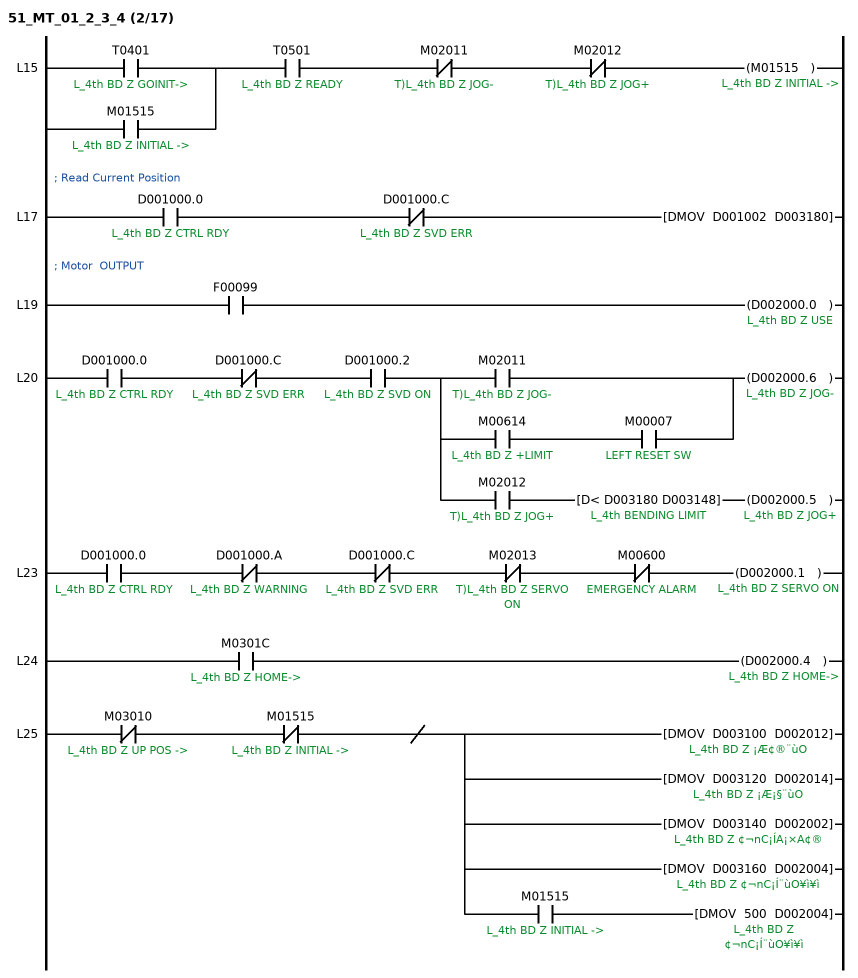
[picture p240: 51_MT_01_2_3_4 rungs L15-L25]
; L15
LOAD      T0401	// L_4th BD Z GOINIT->
OR        M01515	// L_4th BD Z INITIAL ->
AND       T0501	// L_4th BD Z READY
AND NOT   M02011	// T)L_4th BD Z JOG-
AND NOT   M02012	// T)L_4th BD Z JOG+
OUT       M01515	// L_4th BD Z INITIAL ->
; L17
LOAD      D001000.0	// L_4th BD Z CTRL RDY
AND NOT   D001000.C	// L_4th BD Z SVD ERR
DMOV      D001002 D003180
// output comment: Read Current Position
//  Motor  OUTPUT
; L19
LOAD      F00099
OUT       D002000.0	// L_4th BD Z USE
; L20
LOAD      D001000.0	// L_4th BD Z CTRL RDY
AND NOT   D001000.C	// L_4th BD Z SVD ERR
AND       D001000.2	// L_4th BD Z SVD ON
MPUSH
LOAD      M02011	// T)L_4th BD Z JOG-
LOAD      M00614	// L_4th BD Z +LIMIT
AND       M00007	// LEFT RESET SW
OR LOAD
AND LOAD
OUT       D002000.6	// L_4th BD Z JOG-
MPOP
AND       M02012	// T)L_4th BD Z JOG+
ANDD<     D003180 D003148	// L_4th BENDING LIMIT
OUT       D002000.5	// L_4th BD Z JOG+
; L23
LOAD      D001000.0	// L_4th BD Z CTRL RDY
AND NOT   D001000.A	// L_4th BD Z WARNING
AND NOT   D001000.C	// L_4th BD Z SVD ERR
AND NOT   M02013	// T)L_4th BD Z SERVO ON
AND NOT   M00600	// EMERGENCY ALARM
OUT       D002000.1	// L_4th BD Z SERVO ON
; L24
LOAD      M0301C	// L_4th BD Z HOME->
OUT       D002000.4	// L_4th BD Z HOME->
; L25
LOAD NOT  M03010	// L_4th BD Z UP POS ->
AND NOT   M01515	// L_4th BD Z INITIAL ->
NOT
DMOV      D003100 D002012	// L_4th BD Z ¡Æ¢®¨ùO
DMOV      D003120 D002014	// L_4th BD Z ¡Æ¡§¨ùO
DMOV      D003140 D002002	// L_4th BD Z ¢¬nC¡ÍA¡×A¢®
DMOV      D003160 D002004	// L_4th BD Z ¢¬nC¡Í¨ùO¥ì¥ì
AND       M01515	// L_4th BD Z INITIAL ->
DMOV      500 D002004	// L_4th BD Z ¢¬nC¡Í¨ùO¥ì¥ì

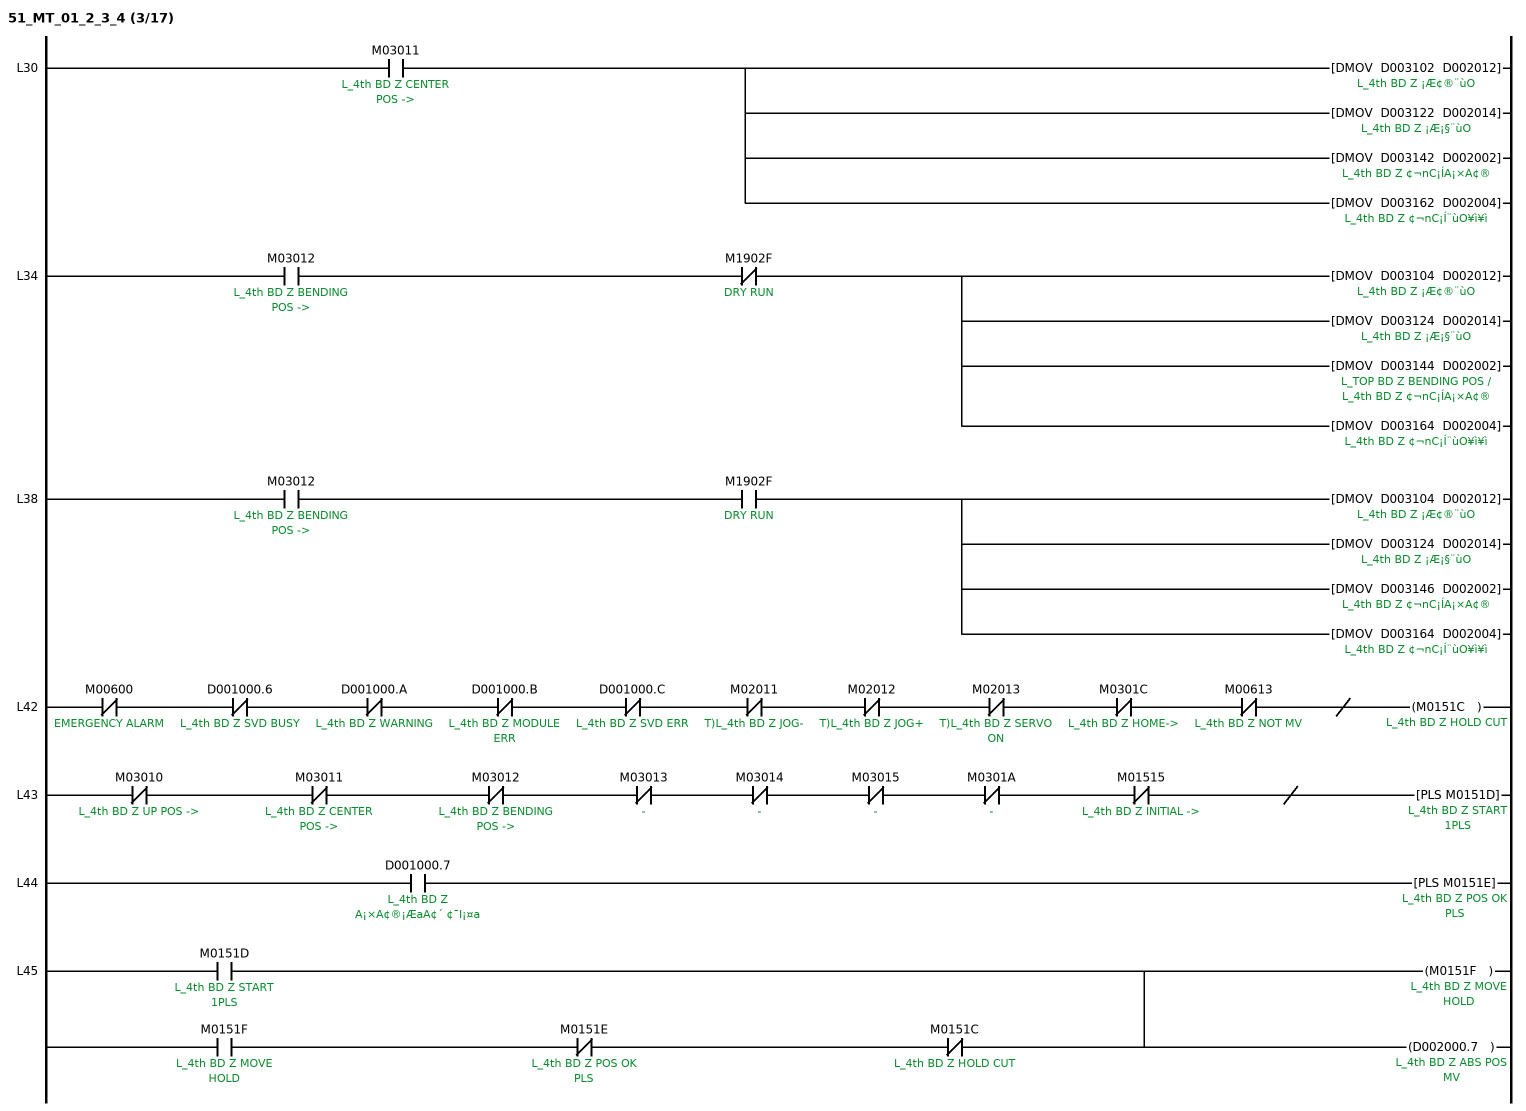
; L30
LOAD      M03011	// L_4th BD Z CENTER POS ->
DMOV      D003102 D002012	// L_4th BD Z ¡Æ¢®¨ùO
DMOV      D003122 D002014	// L_4th BD Z ¡Æ¡§¨ùO
DMOV      D003142 D002002	// L_4th BD Z ¢¬nC¡ÍA¡×A¢®
DMOV      D003162 D002004	// L_4th BD Z ¢¬nC¡Í¨ùO¥ì¥ì
; L34
LOAD      M03012	// L_4th BD Z BENDING POS ->
AND NOT   M1902F	// DRY RUN
DMOV      D003104 D002012	// L_4th BD Z ¡Æ¢®¨ùO
DMOV      D003124 D002014	// L_4th BD Z ¡Æ¡§¨ùO
DMOV      D003144 D002002	// L_TOP BD Z BENDING POS / L_4th BD Z ¢¬nC¡ÍA¡×A¢®
DMOV      D003164 D002004	// L_4th BD Z ¢¬nC¡Í¨ùO¥ì¥ì
; L38
LOAD      M03012	// L_4th BD Z BENDING POS ->
AND       M1902F	// DRY RUN
DMOV      D003104 D002012	// L_4th BD Z ¡Æ¢®¨ùO
DMOV      D003124 D002014	// L_4th BD Z ¡Æ¡§¨ùO
DMOV      D003146 D002002	// L_4th BD Z ¢¬nC¡ÍA¡×A¢®
DMOV      D003164 D002004	// L_4th BD Z ¢¬nC¡Í¨ùO¥ì¥ì
; L42
LOAD NOT  M00600	// EMERGENCY ALARM
AND NOT   D001000.6	// L_4th BD Z SVD BUSY
AND NOT   D001000.A	// L_4th BD Z WARNING
AND NOT   D001000.B	// L_4th BD Z MODULE ERR
AND NOT   D001000.C	// L_4th BD Z SVD ERR
AND NOT   M02011	// T)L_4th BD Z JOG-
AND NOT   M02012	// T)L_4th BD Z JOG+
AND NOT   M02013	// T)L_4th BD Z SERVO ON
AND NOT   M0301C	// L_4th BD Z HOME->
AND NOT   M00613	// L_4th BD Z NOT MV
NOT
OUT       M0151C	// L_4th BD Z HOLD CUT
; L43
LOAD NOT  M03010	// L_4th BD Z UP POS ->
AND NOT   M03011	// L_4th BD Z CENTER POS ->
AND NOT   M03012	// L_4th BD Z BENDING POS ->
AND NOT   M03013	// -
AND NOT   M03014	// -
AND NOT   M03015	// -
AND NOT   M0301A	// -
AND NOT   M01515	// L_4th BD Z INITIAL ->
NOT
OUTP      M0151D	// L_4th BD Z START 1PLS
; L44
LOAD      D001000.7	// L_4th BD Z A¡×A¢®¡ÆaA¢´ ¢¯I¡¤a
OUTP      M0151E	// L_4th BD Z POS OK PLS
; L45
LOAD      M0151D	// L_4th BD Z START 1PLS
LOAD      M0151F	// L_4th BD Z MOVE HOLD
AND NOT   M0151E	// L_4th BD Z POS OK PLS
AND NOT   M0151C	// L_4th BD Z HOLD CUT
OR LOAD
OUT       M0151F	// L_4th BD Z MOVE HOLD
OUT       D002000.7	// L_4th BD Z ABS POS MV

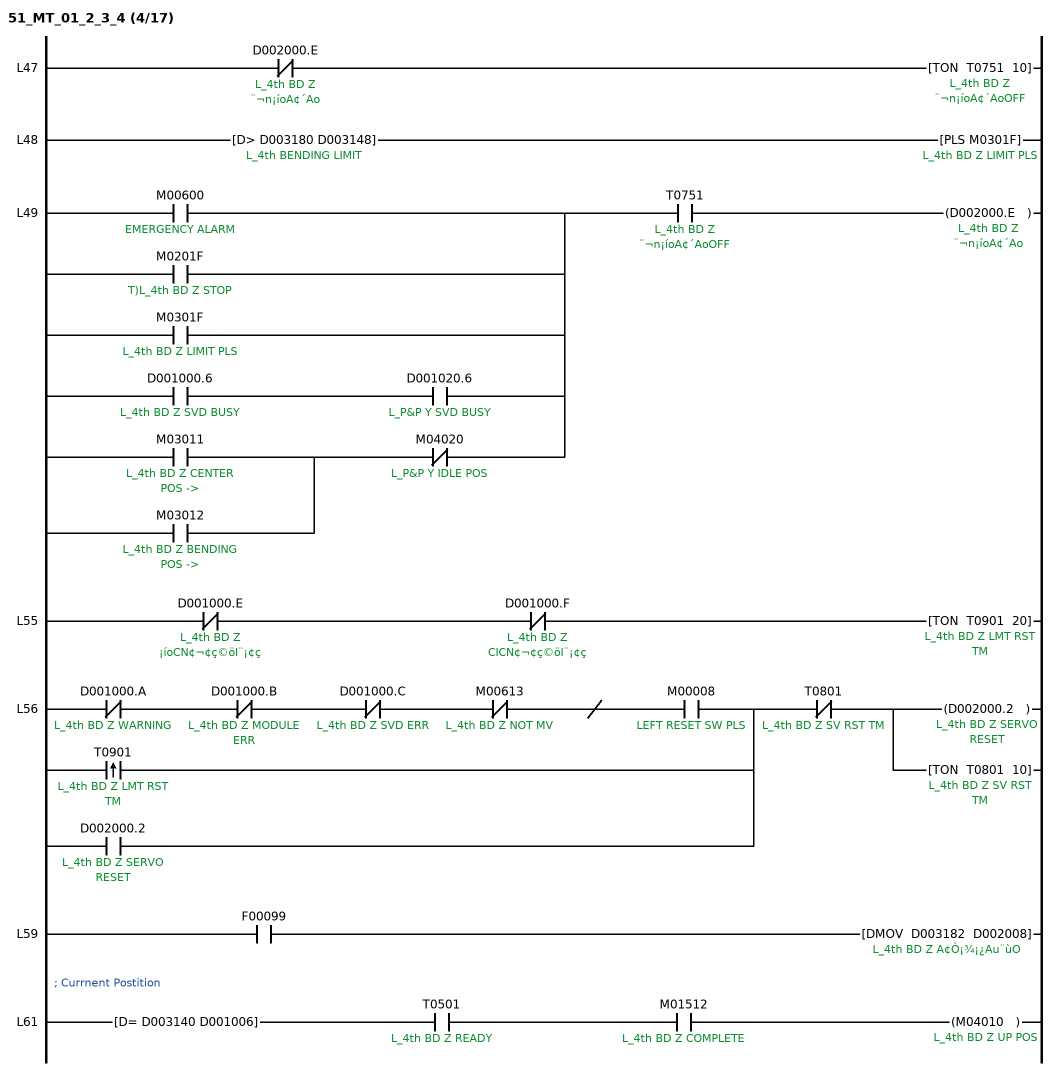
; L47
LOAD NOT  D002000.E	// L_4th BD Z ¨¬n¡íoA¢´Ao
TON       T0751 10	// L_4th BD Z ¨¬n¡íoA¢´AoOFF
; L48
LOADD>    D003180 D003148	// L_4th BENDING LIMIT
OUTP      M0301F	// L_4th BD Z LIMIT PLS
; L49
LOAD      M00600	// EMERGENCY ALARM
OR        M0201F	// T)L_4th BD Z STOP
OR        M0301F	// L_4th BD Z LIMIT PLS
LOAD      D001000.6	// L_4th BD Z SVD BUSY
AND       D001020.6	// L_P&P Y SVD BUSY
OR LOAD
LOAD      M03011	// L_4th BD Z CENTER POS ->
OR        M03012	// L_4th BD Z BENDING POS ->
AND NOT   M04020	// L_P&P Y IDLE POS
OR LOAD
AND       T0751	// L_4th BD Z ¨¬n¡íoA¢´AoOFF
OUT       D002000.E	// L_4th BD Z ¨¬n¡íoA¢´Ao
; L55
LOAD NOT  D001000.E	// L_4th BD Z ¡íoCN¢¬¢ç©öI¨¡¢ç
AND NOT   D001000.F	// L_4th BD Z CICN¢¬¢ç©öI¨¡¢ç
TON       T0901 20	// L_4th BD Z LMT RST TM
; L56
LOAD NOT  D001000.A	// L_4th BD Z WARNING
AND NOT   D001000.B	// L_4th BD Z MODULE ERR
AND NOT   D001000.C	// L_4th BD Z SVD ERR
AND NOT   M00613	// L_4th BD Z NOT MV
NOT
AND       M00008	// LEFT RESET SW PLS
ORP       T0901	// L_4th BD Z LMT RST TM
OR        D002000.2	// L_4th BD Z SERVO RESET
AND NOT   T0801	// L_4th BD Z SV RST TM
OUT       D002000.2	// L_4th BD Z SERVO RESET
TON       T0801 10	// L_4th BD Z SV RST TM
; L59
LOAD      F00099
DMOV      D003182 D002008	// L_4th BD Z A¢Ò¡¾¡¿Au¨ùO
// Currnent Postition
; L61
LOADD=    D003140 D001006
AND       T0501	// L_4th BD Z READY
AND       M01512	// L_4th BD Z COMPLETE
OUT       M04010	// L_4th BD Z UP POS

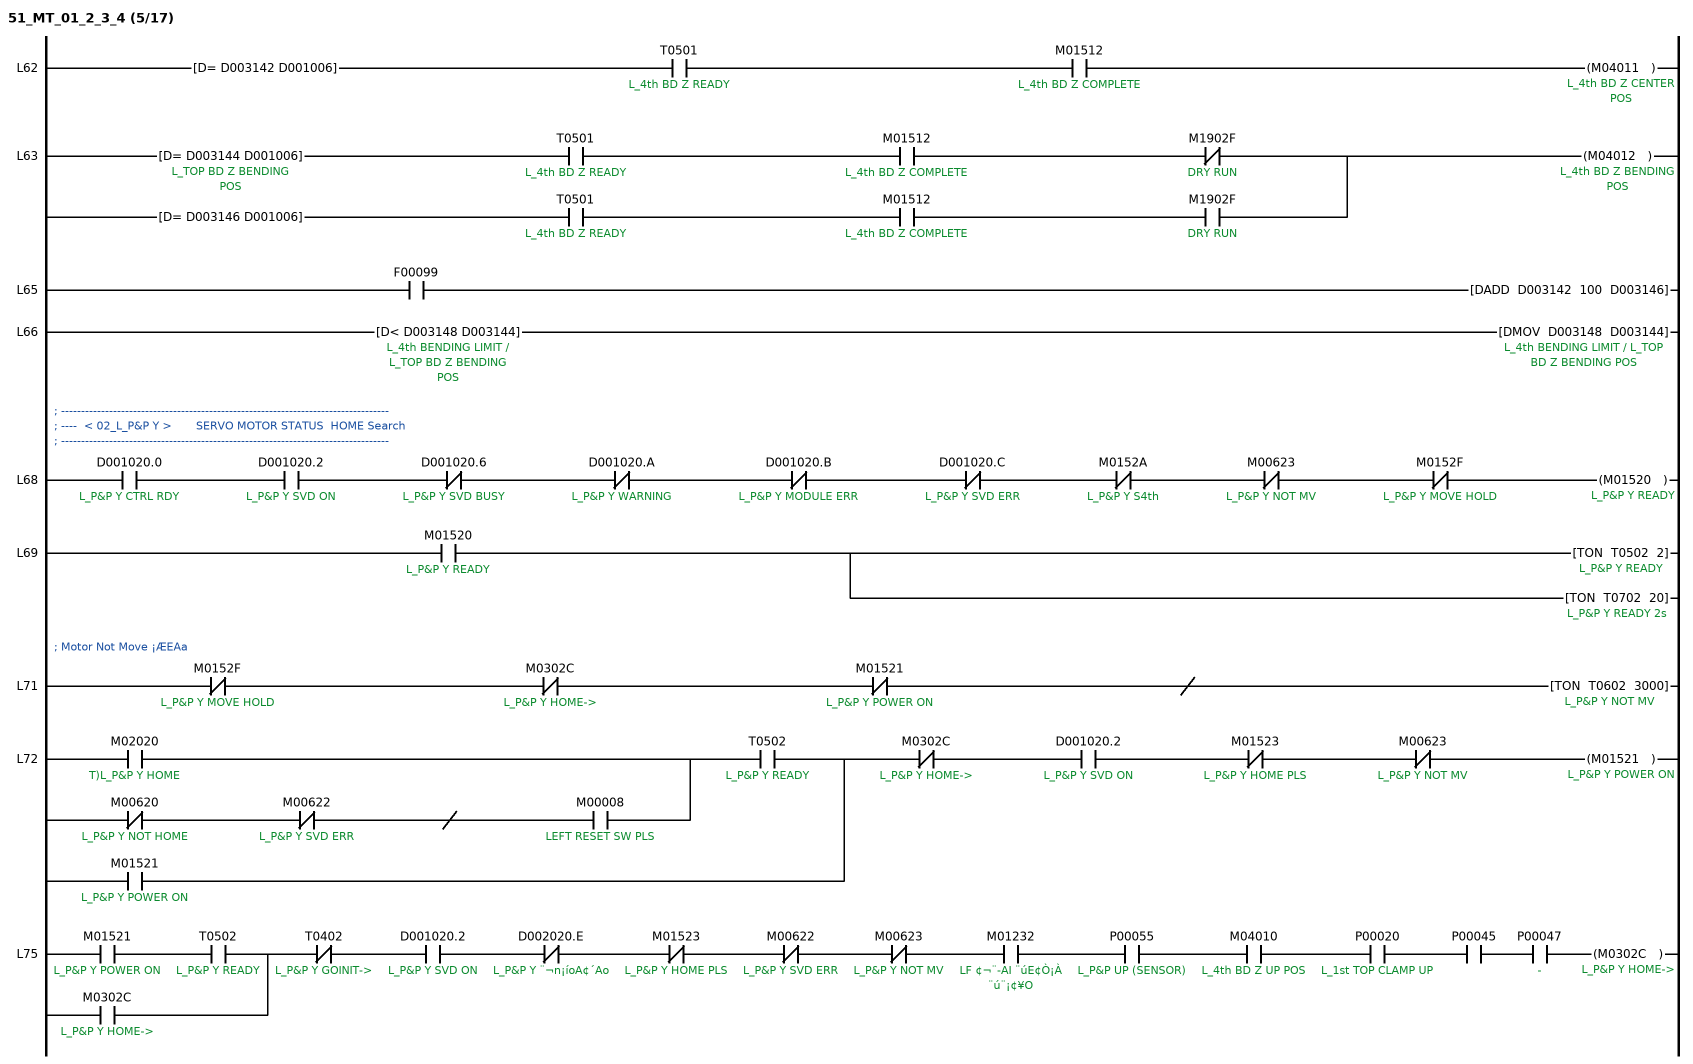
; L62
LOADD=    D003142 D001006
AND       T0501	// L_4th BD Z READY
AND       M01512	// L_4th BD Z COMPLETE
OUT       M04011	// L_4th BD Z CENTER POS
; L63
LOADD=    D003144 D001006	// L_TOP BD Z BENDING POS
AND       T0501	// L_4th BD Z READY
AND       M01512	// L_4th BD Z COMPLETE
AND NOT   M1902F	// DRY RUN
LOADD=    D003146 D001006
AND       T0501	// L_4th BD Z READY
AND       M01512	// L_4th BD Z COMPLETE
AND       M1902F	// DRY RUN
OR LOAD
OUT       M04012	// L_4th BD Z BENDING POS
; L65
LOAD      F00099
DADD      D003142 100 D003146
; L66
LOADD<    D003148 D003144	// L_4th BENDING LIMIT / L_TOP BD Z BENDING POS
DMOV      D003148 D003144	// L_4th BENDING LIMIT / L_TOP BD Z BENDING POS
// ----------------------------------------------------------------------------------
// 
// ----  < 02_L_P&P Y >       SERVO MOTOR STATUS  HOME Search
// 
// ----------------------------------------------------------------------------------
; L68
LOAD      D001020.0	// L_P&P Y CTRL RDY
AND       D001020.2	// L_P&P Y SVD ON
AND NOT   D001020.6	// L_P&P Y SVD BUSY
AND NOT   D001020.A	// L_P&P Y WARNING
AND NOT   D001020.B	// L_P&P Y MODULE ERR
AND NOT   D001020.C	// L_P&P Y SVD ERR
AND NOT   M0152A	// L_P&P Y S4th
AND NOT   M00623	// L_P&P Y NOT MV
AND NOT   M0152F	// L_P&P Y MOVE HOLD
OUT       M01520	// L_P&P Y READY
; L69
LOAD      M01520	// L_P&P Y READY
TON       T0502 2	// L_P&P Y READY
TON       T0702 20	// L_P&P Y READY 2s
; L71
LOAD NOT  M0152F	// L_P&P Y MOVE HOLD
AND NOT   M0302C	// L_P&P Y HOME->
AND NOT   M01521	// L_P&P Y POWER ON
NOT
TON       T0602 3000	// L_P&P Y NOT MV
// output comment: Motor Not Move ¡ÆEAa
; L72
LOAD      M02020	// T)L_P&P Y HOME
LOAD NOT  M00620	// L_P&P Y NOT HOME
AND NOT   M00622	// L_P&P Y SVD ERR
NOT
AND       M00008	// LEFT RESET SW PLS
OR LOAD
AND       T0502	// L_P&P Y READY
OR        M01521	// L_P&P Y POWER ON
AND NOT   M0302C	// L_P&P Y HOME->
AND       D001020.2	// L_P&P Y SVD ON
AND NOT   M01523	// L_P&P Y HOME PLS
AND NOT   M00623	// L_P&P Y NOT MV
OUT       M01521	// L_P&P Y POWER ON
; L75
LOAD      M01521	// L_P&P Y POWER ON
AND       T0502	// L_P&P Y READY
OR        M0302C	// L_P&P Y HOME->
AND NOT   T0402	// L_P&P Y GOINIT->
AND       D001020.2	// L_P&P Y SVD ON
AND NOT   D002020.E	// L_P&P Y ¨¬n¡íoA¢´Ao
AND NOT   M01523	// L_P&P Y HOME PLS
AND NOT   M00622	// L_P&P Y SVD ERR
AND NOT   M00623	// L_P&P Y NOT MV
AND       M01232	// LF ¢¬¨­AI ¨úE¢Ò¡À ¨ú¨¡¢¥O
AND       P00055	// L_P&P UP (SENSOR)
AND       M04010	// L_4th BD Z UP POS
AND       P00020	// L_1st TOP CLAMP UP
AND       P00045
AND       P00047	// -
OUT       M0302C	// L_P&P Y HOME->

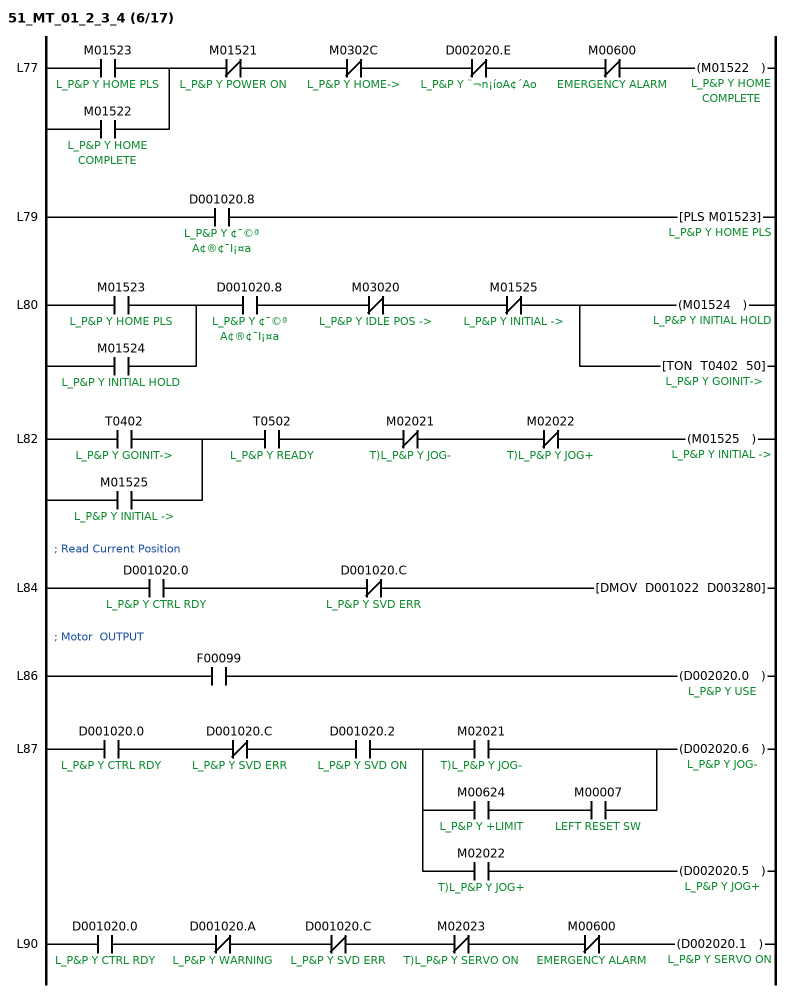
; L77
LOAD      M01523	// L_P&P Y HOME PLS
OR        M01522	// L_P&P Y HOME COMPLETE
AND NOT   M01521	// L_P&P Y POWER ON
AND NOT   M0302C	// L_P&P Y HOME->
AND NOT   D002020.E	// L_P&P Y ¨¬n¡íoA¢´Ao
AND NOT   M00600	// EMERGENCY ALARM
OUT       M01522	// L_P&P Y HOME COMPLETE
; L79
LOAD      D001020.8	// L_P&P Y ¢¯©ªA¢®¢¯I¡¤a
OUTP      M01523	// L_P&P Y HOME PLS
; L80
LOAD      M01523	// L_P&P Y HOME PLS
OR        M01524	// L_P&P Y INITIAL HOLD
AND       D001020.8	// L_P&P Y ¢¯©ªA¢®¢¯I¡¤a
AND NOT   M03020	// L_P&P Y IDLE POS ->
AND NOT   M01525	// L_P&P Y INITIAL ->
OUT       M01524	// L_P&P Y INITIAL HOLD
TON       T0402 50	// L_P&P Y GOINIT->
; L82
LOAD      T0402	// L_P&P Y GOINIT->
OR        M01525	// L_P&P Y INITIAL ->
AND       T0502	// L_P&P Y READY
AND NOT   M02021	// T)L_P&P Y JOG-
AND NOT   M02022	// T)L_P&P Y JOG+
OUT       M01525	// L_P&P Y INITIAL ->
; L84
LOAD      D001020.0	// L_P&P Y CTRL RDY
AND NOT   D001020.C	// L_P&P Y SVD ERR
DMOV      D001022 D003280
// output comment: Read Current Position
//  Motor  OUTPUT
; L86
LOAD      F00099
OUT       D002020.0	// L_P&P Y USE
; L87
LOAD      D001020.0	// L_P&P Y CTRL RDY
AND NOT   D001020.C	// L_P&P Y SVD ERR
AND       D001020.2	// L_P&P Y SVD ON
MPUSH
LOAD      M02021	// T)L_P&P Y JOG-
LOAD      M00624	// L_P&P Y +LIMIT
AND       M00007	// LEFT RESET SW
OR LOAD
AND LOAD
OUT       D002020.6	// L_P&P Y JOG-
MPOP
AND       M02022	// T)L_P&P Y JOG+
OUT       D002020.5	// L_P&P Y JOG+
; L90
LOAD      D001020.0	// L_P&P Y CTRL RDY
AND NOT   D001020.A	// L_P&P Y WARNING
AND NOT   D001020.C	// L_P&P Y SVD ERR
AND NOT   M02023	// T)L_P&P Y SERVO ON
AND NOT   M00600	// EMERGENCY ALARM
OUT       D002020.1	// L_P&P Y SERVO ON

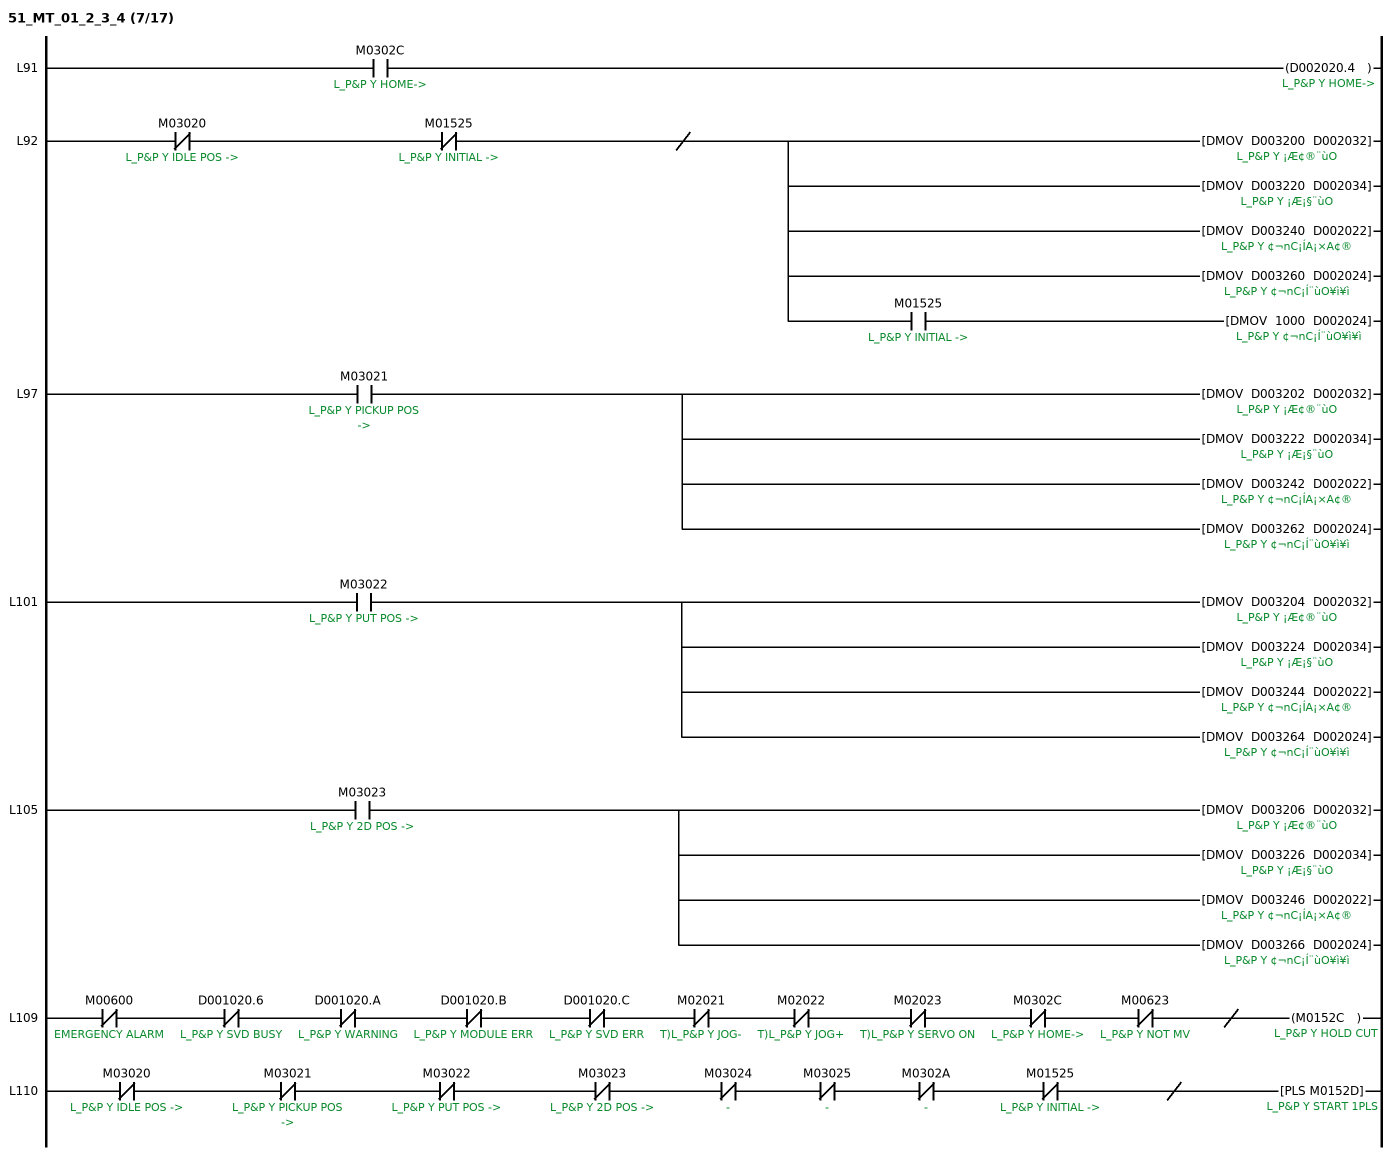
; L91
LOAD      M0302C	// L_P&P Y HOME->
OUT       D002020.4	// L_P&P Y HOME->
; L92
LOAD NOT  M03020	// L_P&P Y IDLE POS ->
AND NOT   M01525	// L_P&P Y INITIAL ->
NOT
DMOV      D003200 D002032	// L_P&P Y ¡Æ¢®¨ùO
DMOV      D003220 D002034	// L_P&P Y ¡Æ¡§¨ùO
DMOV      D003240 D002022	// L_P&P Y ¢¬nC¡ÍA¡×A¢®
DMOV      D003260 D002024	// L_P&P Y ¢¬nC¡Í¨ùO¥ì¥ì
AND       M01525	// L_P&P Y INITIAL ->
DMOV      1000 D002024	// L_P&P Y ¢¬nC¡Í¨ùO¥ì¥ì
; L97
LOAD      M03021	// L_P&P Y PICKUP POS ->
DMOV      D003202 D002032	// L_P&P Y ¡Æ¢®¨ùO
DMOV      D003222 D002034	// L_P&P Y ¡Æ¡§¨ùO
DMOV      D003242 D002022	// L_P&P Y ¢¬nC¡ÍA¡×A¢®
DMOV      D003262 D002024	// L_P&P Y ¢¬nC¡Í¨ùO¥ì¥ì
; L101
LOAD      M03022	// L_P&P Y PUT POS ->
DMOV      D003204 D002032	// L_P&P Y ¡Æ¢®¨ùO
DMOV      D003224 D002034	// L_P&P Y ¡Æ¡§¨ùO
DMOV      D003244 D002022	// L_P&P Y ¢¬nC¡ÍA¡×A¢®
DMOV      D003264 D002024	// L_P&P Y ¢¬nC¡Í¨ùO¥ì¥ì
; L105
LOAD      M03023	// L_P&P Y 2D POS ->
DMOV      D003206 D002032	// L_P&P Y ¡Æ¢®¨ùO
DMOV      D003226 D002034	// L_P&P Y ¡Æ¡§¨ùO
DMOV      D003246 D002022	// L_P&P Y ¢¬nC¡ÍA¡×A¢®
DMOV      D003266 D002024	// L_P&P Y ¢¬nC¡Í¨ùO¥ì¥ì
; L109
LOAD NOT  M00600	// EMERGENCY ALARM
AND NOT   D001020.6	// L_P&P Y SVD BUSY
AND NOT   D001020.A	// L_P&P Y WARNING
AND NOT   D001020.B	// L_P&P Y MODULE ERR
AND NOT   D001020.C	// L_P&P Y SVD ERR
AND NOT   M02021	// T)L_P&P Y JOG-
AND NOT   M02022	// T)L_P&P Y JOG+
AND NOT   M02023	// T)L_P&P Y SERVO ON
AND NOT   M0302C	// L_P&P Y HOME->
AND NOT   M00623	// L_P&P Y NOT MV
NOT
OUT       M0152C	// L_P&P Y HOLD CUT
; L110
LOAD NOT  M03020	// L_P&P Y IDLE POS ->
AND NOT   M03021	// L_P&P Y PICKUP POS ->
AND NOT   M03022	// L_P&P Y PUT POS ->
AND NOT   M03023	// L_P&P Y 2D POS ->
AND NOT   M03024	// -
AND NOT   M03025	// -
AND NOT   M0302A	// -
AND NOT   M01525	// L_P&P Y INITIAL ->
NOT
OUTP      M0152D	// L_P&P Y START 1PLS

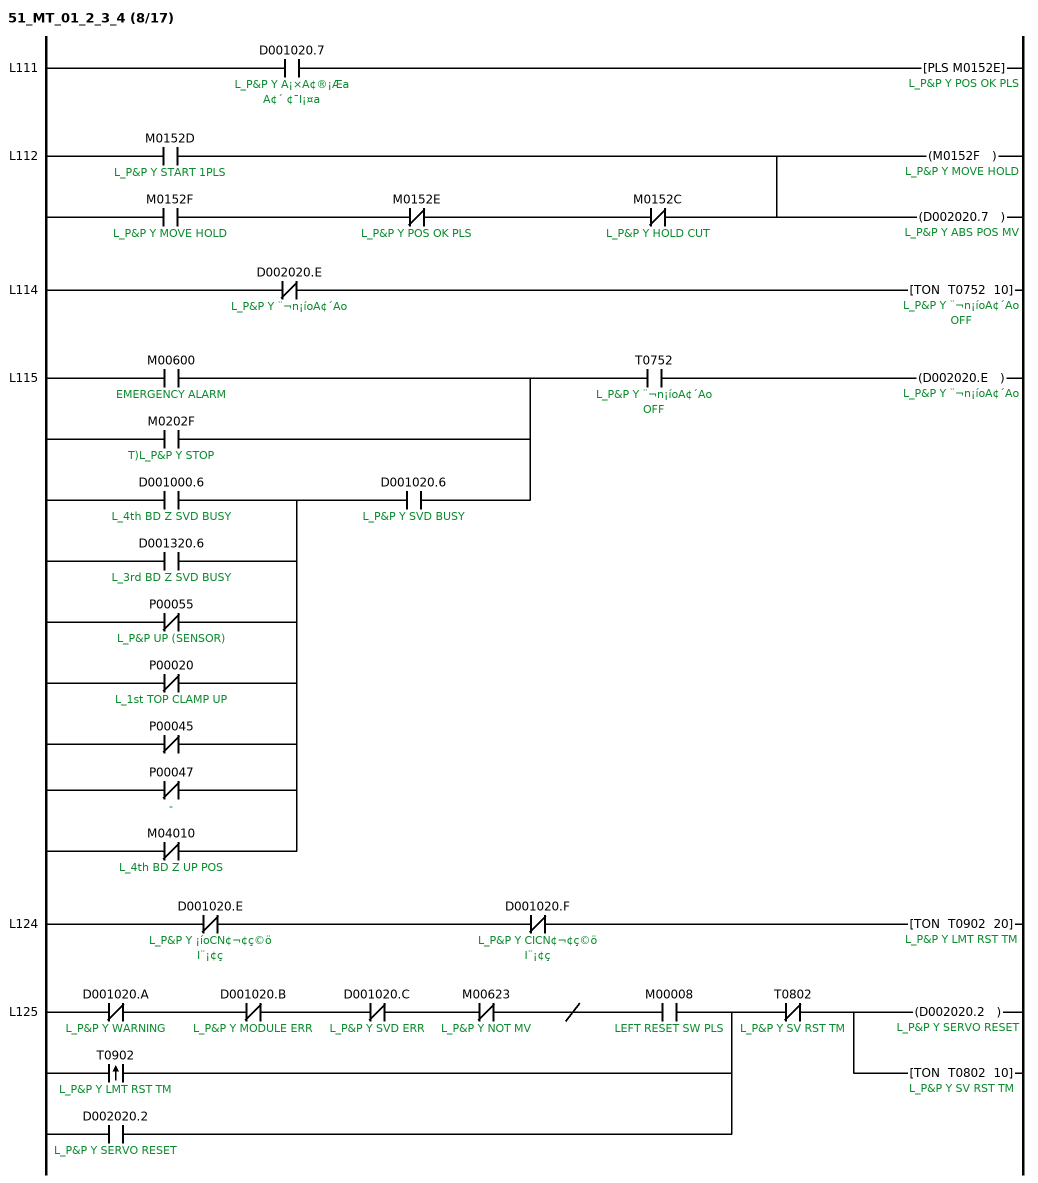
; L111
LOAD      D001020.7	// L_P&P Y A¡×A¢®¡ÆaA¢´ ¢¯I¡¤a
OUTP      M0152E	// L_P&P Y POS OK PLS
; L112
LOAD      M0152D	// L_P&P Y START 1PLS
LOAD      M0152F	// L_P&P Y MOVE HOLD
AND NOT   M0152E	// L_P&P Y POS OK PLS
AND NOT   M0152C	// L_P&P Y HOLD CUT
OR LOAD
OUT       M0152F	// L_P&P Y MOVE HOLD
OUT       D002020.7	// L_P&P Y ABS POS MV
; L114
LOAD NOT  D002020.E	// L_P&P Y ¨¬n¡íoA¢´Ao
TON       T0752 10	// L_P&P Y ¨¬n¡íoA¢´AoOFF
; L115
LOAD      M00600	// EMERGENCY ALARM
OR        M0202F	// T)L_P&P Y STOP
LOAD      D001000.6	// L_4th BD Z SVD BUSY
OR        D001320.6	// L_3rd BD Z SVD BUSY
OR NOT    P00055	// L_P&P UP (SENSOR)
OR NOT    P00020	// L_1st TOP CLAMP UP
OR NOT    P00045
OR NOT    P00047	// -
OR NOT    M04010	// L_4th BD Z UP POS
AND       D001020.6	// L_P&P Y SVD BUSY
OR LOAD
AND       T0752	// L_P&P Y ¨¬n¡íoA¢´AoOFF
OUT       D002020.E	// L_P&P Y ¨¬n¡íoA¢´Ao
; L124
LOAD NOT  D001020.E	// L_P&P Y ¡íoCN¢¬¢ç©öI¨¡¢ç
AND NOT   D001020.F	// L_P&P Y CICN¢¬¢ç©öI¨¡¢ç
TON       T0902 20	// L_P&P Y LMT RST TM
; L125
LOAD NOT  D001020.A	// L_P&P Y WARNING
AND NOT   D001020.B	// L_P&P Y MODULE ERR
AND NOT   D001020.C	// L_P&P Y SVD ERR
AND NOT   M00623	// L_P&P Y NOT MV
NOT
AND       M00008	// LEFT RESET SW PLS
ORP       T0902	// L_P&P Y LMT RST TM
OR        D002020.2	// L_P&P Y SERVO RESET
AND NOT   T0802	// L_P&P Y SV RST TM
OUT       D002020.2	// L_P&P Y SERVO RESET
TON       T0802 10	// L_P&P Y SV RST TM

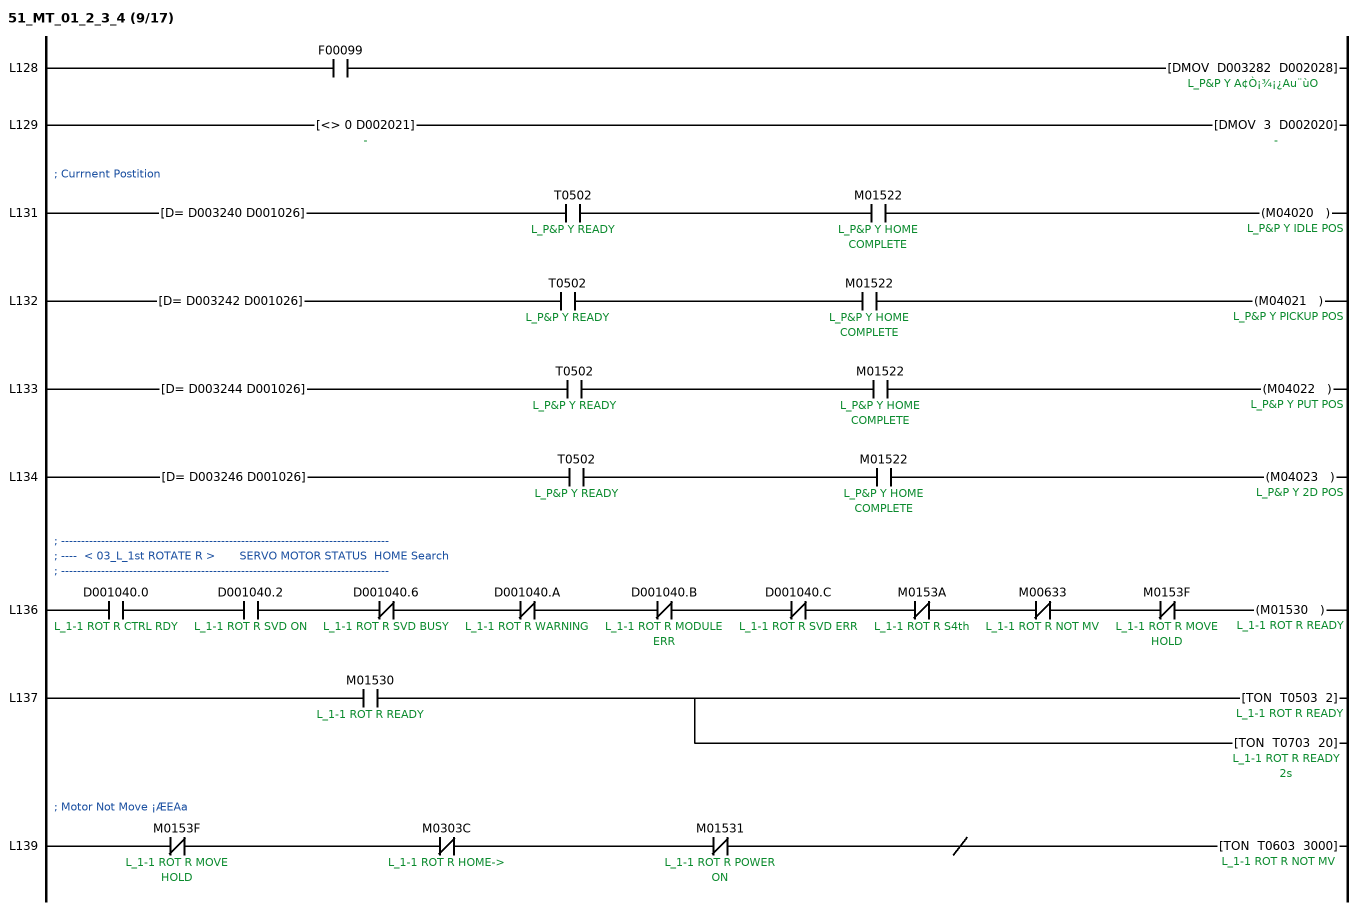
; L128
LOAD      F00099
DMOV      D003282 D002028	// L_P&P Y A¢Ò¡¾¡¿Au¨ùO
; L129
LOAD<>    0 D002021	// -
DMOV      3 D002020	// -
// Currnent Postition
; L131
LOADD=    D003240 D001026
AND       T0502	// L_P&P Y READY
AND       M01522	// L_P&P Y HOME COMPLETE
OUT       M04020	// L_P&P Y IDLE POS
; L132
LOADD=    D003242 D001026
AND       T0502	// L_P&P Y READY
AND       M01522	// L_P&P Y HOME COMPLETE
OUT       M04021	// L_P&P Y PICKUP POS
; L133
LOADD=    D003244 D001026
AND       T0502	// L_P&P Y READY
AND       M01522	// L_P&P Y HOME COMPLETE
OUT       M04022	// L_P&P Y PUT POS
; L134
LOADD=    D003246 D001026
AND       T0502	// L_P&P Y READY
AND       M01522	// L_P&P Y HOME COMPLETE
OUT       M04023	// L_P&P Y 2D POS
// ----------------------------------------------------------------------------------
// 
// ----  < 03_L_1st ROTATE R >       SERVO MOTOR STATUS  HOME Search
// 
// ----------------------------------------------------------------------------------
; L136
LOAD      D001040.0	// L_1-1 ROT R CTRL RDY
AND       D001040.2	// L_1-1 ROT R SVD ON
AND NOT   D001040.6	// L_1-1 ROT R SVD BUSY
AND NOT   D001040.A	// L_1-1 ROT R WARNING
AND NOT   D001040.B	// L_1-1 ROT R MODULE ERR
AND NOT   D001040.C	// L_1-1 ROT R SVD ERR
AND NOT   M0153A	// L_1-1 ROT R S4th
AND NOT   M00633	// L_1-1 ROT R NOT MV
AND NOT   M0153F	// L_1-1 ROT R MOVE HOLD
OUT       M01530	// L_1-1 ROT R READY
; L137
LOAD      M01530	// L_1-1 ROT R READY
TON       T0503 2	// L_1-1 ROT R READY
TON       T0703 20	// L_1-1 ROT R READY 2s
; L139
LOAD NOT  M0153F	// L_1-1 ROT R MOVE HOLD
AND NOT   M0303C	// L_1-1 ROT R HOME->
AND NOT   M01531	// L_1-1 ROT R POWER ON
NOT
TON       T0603 3000	// L_1-1 ROT R NOT MV
// output comment: Motor Not Move ¡ÆEAa

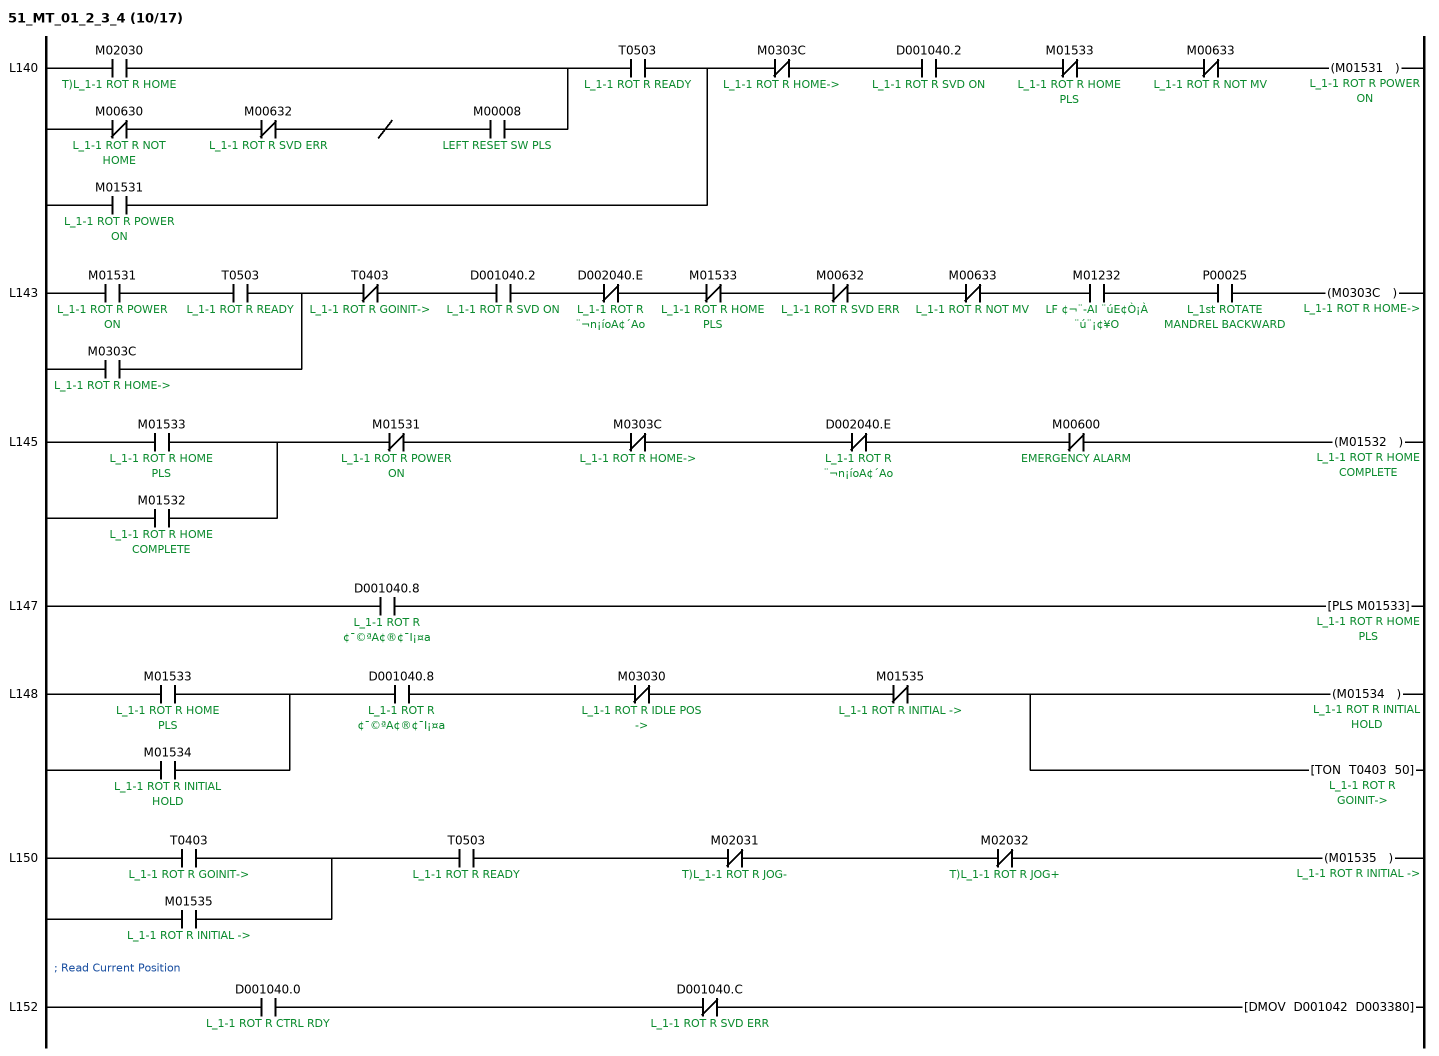
; L140
LOAD      M02030	// T)L_1-1 ROT R HOME
LOAD NOT  M00630	// L_1-1 ROT R NOT HOME
AND NOT   M00632	// L_1-1 ROT R SVD ERR
NOT
AND       M00008	// LEFT RESET SW PLS
OR LOAD
AND       T0503	// L_1-1 ROT R READY
OR        M01531	// L_1-1 ROT R POWER ON
AND NOT   M0303C	// L_1-1 ROT R HOME->
AND       D001040.2	// L_1-1 ROT R SVD ON
AND NOT   M01533	// L_1-1 ROT R HOME PLS
AND NOT   M00633	// L_1-1 ROT R NOT MV
OUT       M01531	// L_1-1 ROT R POWER ON
; L143
LOAD      M01531	// L_1-1 ROT R POWER ON
AND       T0503	// L_1-1 ROT R READY
OR        M0303C	// L_1-1 ROT R HOME->
AND NOT   T0403	// L_1-1 ROT R GOINIT->
AND       D001040.2	// L_1-1 ROT R SVD ON
AND NOT   D002040.E	// L_1-1 ROT R ¨¬n¡íoA¢´Ao
AND NOT   M01533	// L_1-1 ROT R HOME PLS
AND NOT   M00632	// L_1-1 ROT R SVD ERR
AND NOT   M00633	// L_1-1 ROT R NOT MV
AND       M01232	// LF ¢¬¨­AI ¨úE¢Ò¡À ¨ú¨¡¢¥O
AND       P00025	// L_1st ROTATE MANDREL BACKWARD
OUT       M0303C	// L_1-1 ROT R HOME->
; L145
LOAD      M01533	// L_1-1 ROT R HOME PLS
OR        M01532	// L_1-1 ROT R HOME COMPLETE
AND NOT   M01531	// L_1-1 ROT R POWER ON
AND NOT   M0303C	// L_1-1 ROT R HOME->
AND NOT   D002040.E	// L_1-1 ROT R ¨¬n¡íoA¢´Ao
AND NOT   M00600	// EMERGENCY ALARM
OUT       M01532	// L_1-1 ROT R HOME COMPLETE
; L147
LOAD      D001040.8	// L_1-1 ROT R ¢¯©ªA¢®¢¯I¡¤a
OUTP      M01533	// L_1-1 ROT R HOME PLS
; L148
LOAD      M01533	// L_1-1 ROT R HOME PLS
OR        M01534	// L_1-1 ROT R INITIAL HOLD
AND       D001040.8	// L_1-1 ROT R ¢¯©ªA¢®¢¯I¡¤a
AND NOT   M03030	// L_1-1 ROT R IDLE POS ->
AND NOT   M01535	// L_1-1 ROT R INITIAL ->
OUT       M01534	// L_1-1 ROT R INITIAL HOLD
TON       T0403 50	// L_1-1 ROT R GOINIT->
; L150
LOAD      T0403	// L_1-1 ROT R GOINIT->
OR        M01535	// L_1-1 ROT R INITIAL ->
AND       T0503	// L_1-1 ROT R READY
AND NOT   M02031	// T)L_1-1 ROT R JOG-
AND NOT   M02032	// T)L_1-1 ROT R JOG+
OUT       M01535	// L_1-1 ROT R INITIAL ->
; L152
LOAD      D001040.0	// L_1-1 ROT R CTRL RDY
AND NOT   D001040.C	// L_1-1 ROT R SVD ERR
DMOV      D001042 D003380
// output comment: Read Current Position

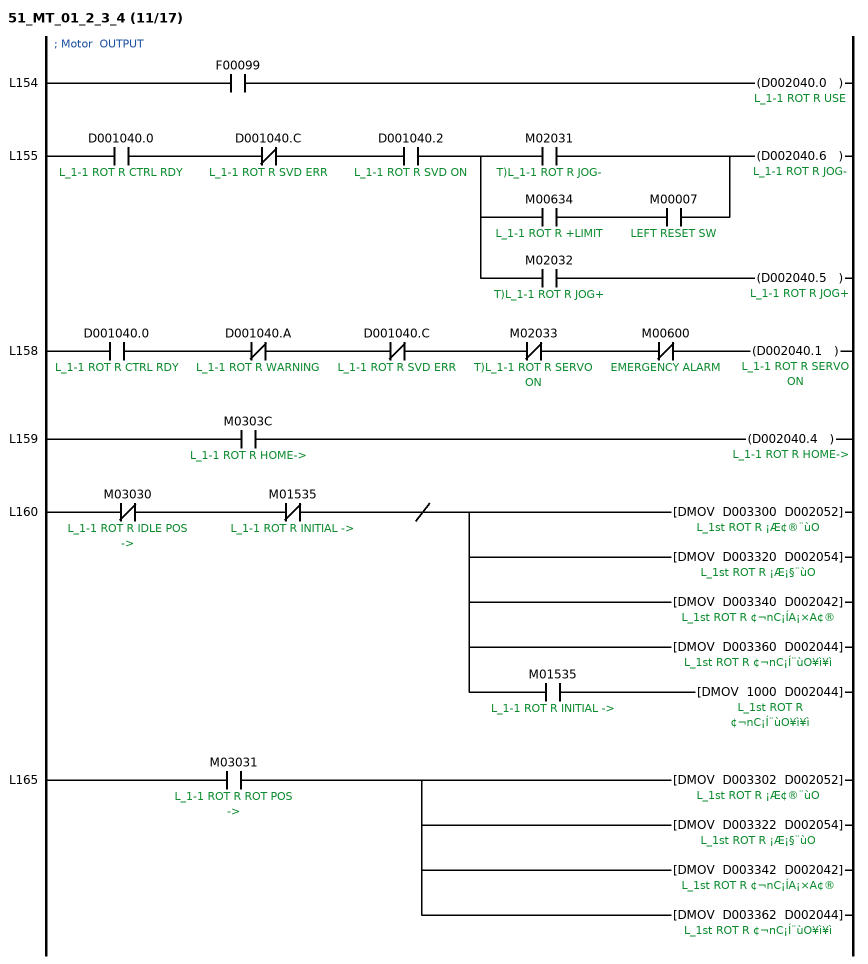
//  Motor  OUTPUT
; L154
LOAD      F00099
OUT       D002040.0	// L_1-1 ROT R USE
; L155
LOAD      D001040.0	// L_1-1 ROT R CTRL RDY
AND NOT   D001040.C	// L_1-1 ROT R SVD ERR
AND       D001040.2	// L_1-1 ROT R SVD ON
MPUSH
LOAD      M02031	// T)L_1-1 ROT R JOG-
LOAD      M00634	// L_1-1 ROT R +LIMIT
AND       M00007	// LEFT RESET SW
OR LOAD
AND LOAD
OUT       D002040.6	// L_1-1 ROT R JOG-
MPOP
AND       M02032	// T)L_1-1 ROT R JOG+
OUT       D002040.5	// L_1-1 ROT R JOG+
; L158
LOAD      D001040.0	// L_1-1 ROT R CTRL RDY
AND NOT   D001040.A	// L_1-1 ROT R WARNING
AND NOT   D001040.C	// L_1-1 ROT R SVD ERR
AND NOT   M02033	// T)L_1-1 ROT R SERVO ON
AND NOT   M00600	// EMERGENCY ALARM
OUT       D002040.1	// L_1-1 ROT R SERVO ON
; L159
LOAD      M0303C	// L_1-1 ROT R HOME->
OUT       D002040.4	// L_1-1 ROT R HOME->
; L160
LOAD NOT  M03030	// L_1-1 ROT R IDLE POS ->
AND NOT   M01535	// L_1-1 ROT R INITIAL ->
NOT
DMOV      D003300 D002052	// L_1st ROT R ¡Æ¢®¨ùO
DMOV      D003320 D002054	// L_1st ROT R ¡Æ¡§¨ùO
DMOV      D003340 D002042	// L_1st ROT R ¢¬nC¡ÍA¡×A¢®
DMOV      D003360 D002044	// L_1st ROT R ¢¬nC¡Í¨ùO¥ì¥ì
AND       M01535	// L_1-1 ROT R INITIAL ->
DMOV      1000 D002044	// L_1st ROT R ¢¬nC¡Í¨ùO¥ì¥ì
; L165
LOAD      M03031	// L_1-1 ROT R ROT POS ->
DMOV      D003302 D002052	// L_1st ROT R ¡Æ¢®¨ùO
DMOV      D003322 D002054	// L_1st ROT R ¡Æ¡§¨ùO
DMOV      D003342 D002042	// L_1st ROT R ¢¬nC¡ÍA¡×A¢®
DMOV      D003362 D002044	// L_1st ROT R ¢¬nC¡Í¨ùO¥ì¥ì

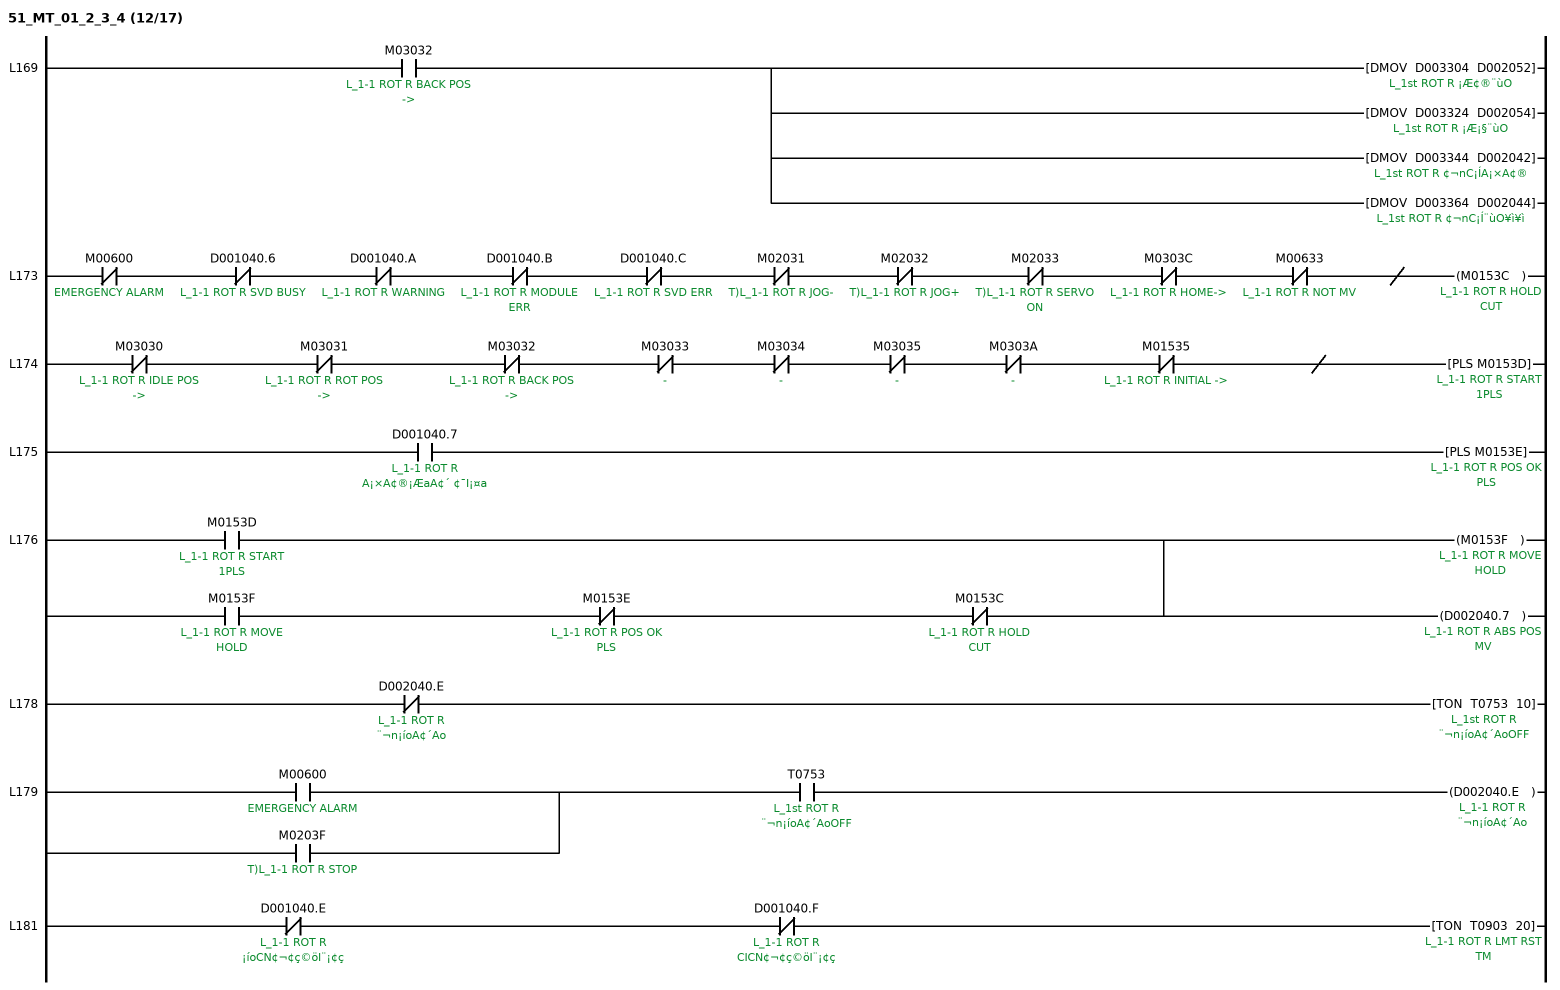
; L169
LOAD      M03032	// L_1-1 ROT R BACK POS ->
DMOV      D003304 D002052	// L_1st ROT R ¡Æ¢®¨ùO
DMOV      D003324 D002054	// L_1st ROT R ¡Æ¡§¨ùO
DMOV      D003344 D002042	// L_1st ROT R ¢¬nC¡ÍA¡×A¢®
DMOV      D003364 D002044	// L_1st ROT R ¢¬nC¡Í¨ùO¥ì¥ì
; L173
LOAD NOT  M00600	// EMERGENCY ALARM
AND NOT   D001040.6	// L_1-1 ROT R SVD BUSY
AND NOT   D001040.A	// L_1-1 ROT R WARNING
AND NOT   D001040.B	// L_1-1 ROT R MODULE ERR
AND NOT   D001040.C	// L_1-1 ROT R SVD ERR
AND NOT   M02031	// T)L_1-1 ROT R JOG-
AND NOT   M02032	// T)L_1-1 ROT R JOG+
AND NOT   M02033	// T)L_1-1 ROT R SERVO ON
AND NOT   M0303C	// L_1-1 ROT R HOME->
AND NOT   M00633	// L_1-1 ROT R NOT MV
NOT
OUT       M0153C	// L_1-1 ROT R HOLD CUT
; L174
LOAD NOT  M03030	// L_1-1 ROT R IDLE POS ->
AND NOT   M03031	// L_1-1 ROT R ROT POS ->
AND NOT   M03032	// L_1-1 ROT R BACK POS ->
AND NOT   M03033	// -
AND NOT   M03034	// -
AND NOT   M03035	// -
AND NOT   M0303A	// -
AND NOT   M01535	// L_1-1 ROT R INITIAL ->
NOT
OUTP      M0153D	// L_1-1 ROT R START 1PLS
; L175
LOAD      D001040.7	// L_1-1 ROT R A¡×A¢®¡ÆaA¢´ ¢¯I¡¤a
OUTP      M0153E	// L_1-1 ROT R POS OK PLS
; L176
LOAD      M0153D	// L_1-1 ROT R START 1PLS
LOAD      M0153F	// L_1-1 ROT R MOVE HOLD
AND NOT   M0153E	// L_1-1 ROT R POS OK PLS
AND NOT   M0153C	// L_1-1 ROT R HOLD CUT
OR LOAD
OUT       M0153F	// L_1-1 ROT R MOVE HOLD
OUT       D002040.7	// L_1-1 ROT R ABS POS MV
; L178
LOAD NOT  D002040.E	// L_1-1 ROT R ¨¬n¡íoA¢´Ao
TON       T0753 10	// L_1st ROT R ¨¬n¡íoA¢´AoOFF
; L179
LOAD      M00600	// EMERGENCY ALARM
OR        M0203F	// T)L_1-1 ROT R STOP
AND       T0753	// L_1st ROT R ¨¬n¡íoA¢´AoOFF
OUT       D002040.E	// L_1-1 ROT R ¨¬n¡íoA¢´Ao
; L181
LOAD NOT  D001040.E	// L_1-1 ROT R ¡íoCN¢¬¢ç©öI¨¡¢ç
AND NOT   D001040.F	// L_1-1 ROT R CICN¢¬¢ç©öI¨¡¢ç
TON       T0903 20	// L_1-1 ROT R LMT RST TM

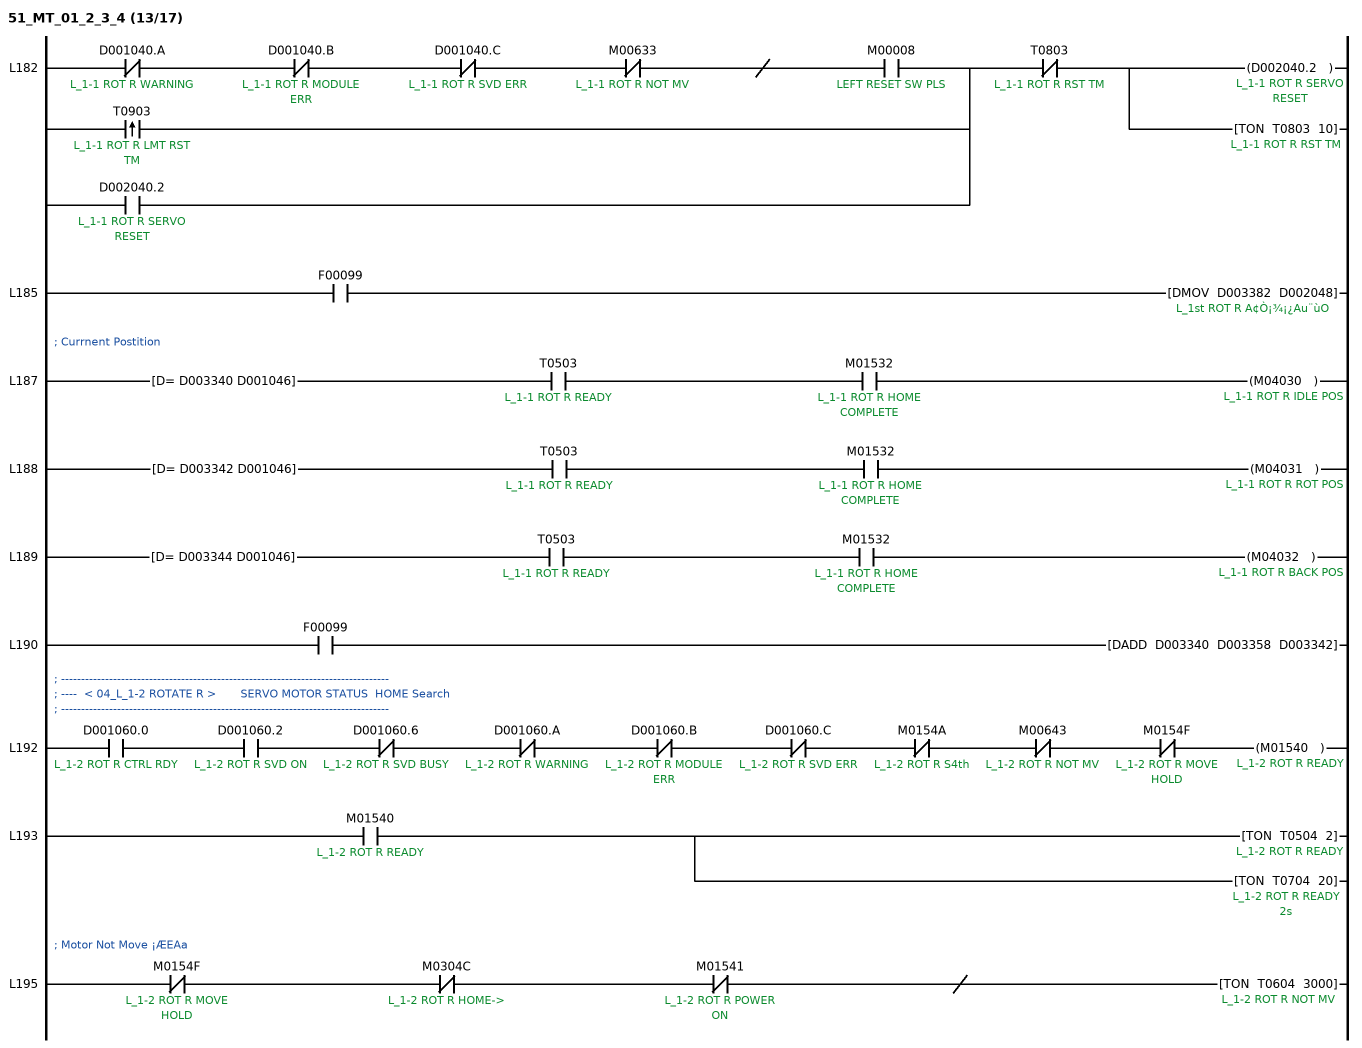
; L182
LOAD NOT  D001040.A	// L_1-1 ROT R WARNING
AND NOT   D001040.B	// L_1-1 ROT R MODULE ERR
AND NOT   D001040.C	// L_1-1 ROT R SVD ERR
AND NOT   M00633	// L_1-1 ROT R NOT MV
NOT
AND       M00008	// LEFT RESET SW PLS
ORP       T0903	// L_1-1 ROT R LMT RST TM
OR        D002040.2	// L_1-1 ROT R SERVO RESET
AND NOT   T0803	// L_1-1 ROT R RST TM
OUT       D002040.2	// L_1-1 ROT R SERVO RESET
TON       T0803 10	// L_1-1 ROT R RST TM
; L185
LOAD      F00099
DMOV      D003382 D002048	// L_1st ROT R A¢Ò¡¾¡¿Au¨ùO
// Currnent Postition
; L187
LOADD=    D003340 D001046
AND       T0503	// L_1-1 ROT R READY
AND       M01532	// L_1-1 ROT R HOME COMPLETE
OUT       M04030	// L_1-1 ROT R IDLE POS
; L188
LOADD=    D003342 D001046
AND       T0503	// L_1-1 ROT R READY
AND       M01532	// L_1-1 ROT R HOME COMPLETE
OUT       M04031	// L_1-1 ROT R ROT POS
; L189
LOADD=    D003344 D001046
AND       T0503	// L_1-1 ROT R READY
AND       M01532	// L_1-1 ROT R HOME COMPLETE
OUT       M04032	// L_1-1 ROT R BACK POS
; L190
LOAD      F00099
DADD      D003340 D003358 D003342
// ----------------------------------------------------------------------------------
// 
// ----  < 04_L_1-2 ROTATE R >       SERVO MOTOR STATUS  HOME Search
// 
// ----------------------------------------------------------------------------------
; L192
LOAD      D001060.0	// L_1-2 ROT R CTRL RDY
AND       D001060.2	// L_1-2 ROT R SVD ON
AND NOT   D001060.6	// L_1-2 ROT R SVD BUSY
AND NOT   D001060.A	// L_1-2 ROT R WARNING
AND NOT   D001060.B	// L_1-2 ROT R MODULE ERR
AND NOT   D001060.C	// L_1-2 ROT R SVD ERR
AND NOT   M0154A	// L_1-2 ROT R S4th
AND NOT   M00643	// L_1-2 ROT R NOT MV
AND NOT   M0154F	// L_1-2 ROT R MOVE HOLD
OUT       M01540	// L_1-2 ROT R READY
; L193
LOAD      M01540	// L_1-2 ROT R READY
TON       T0504 2	// L_1-2 ROT R READY
TON       T0704 20	// L_1-2 ROT R READY 2s
; L195
LOAD NOT  M0154F	// L_1-2 ROT R MOVE HOLD
AND NOT   M0304C	// L_1-2 ROT R HOME->
AND NOT   M01541	// L_1-2 ROT R POWER ON
NOT
TON       T0604 3000	// L_1-2 ROT R NOT MV
// output comment: Motor Not Move ¡ÆEAa

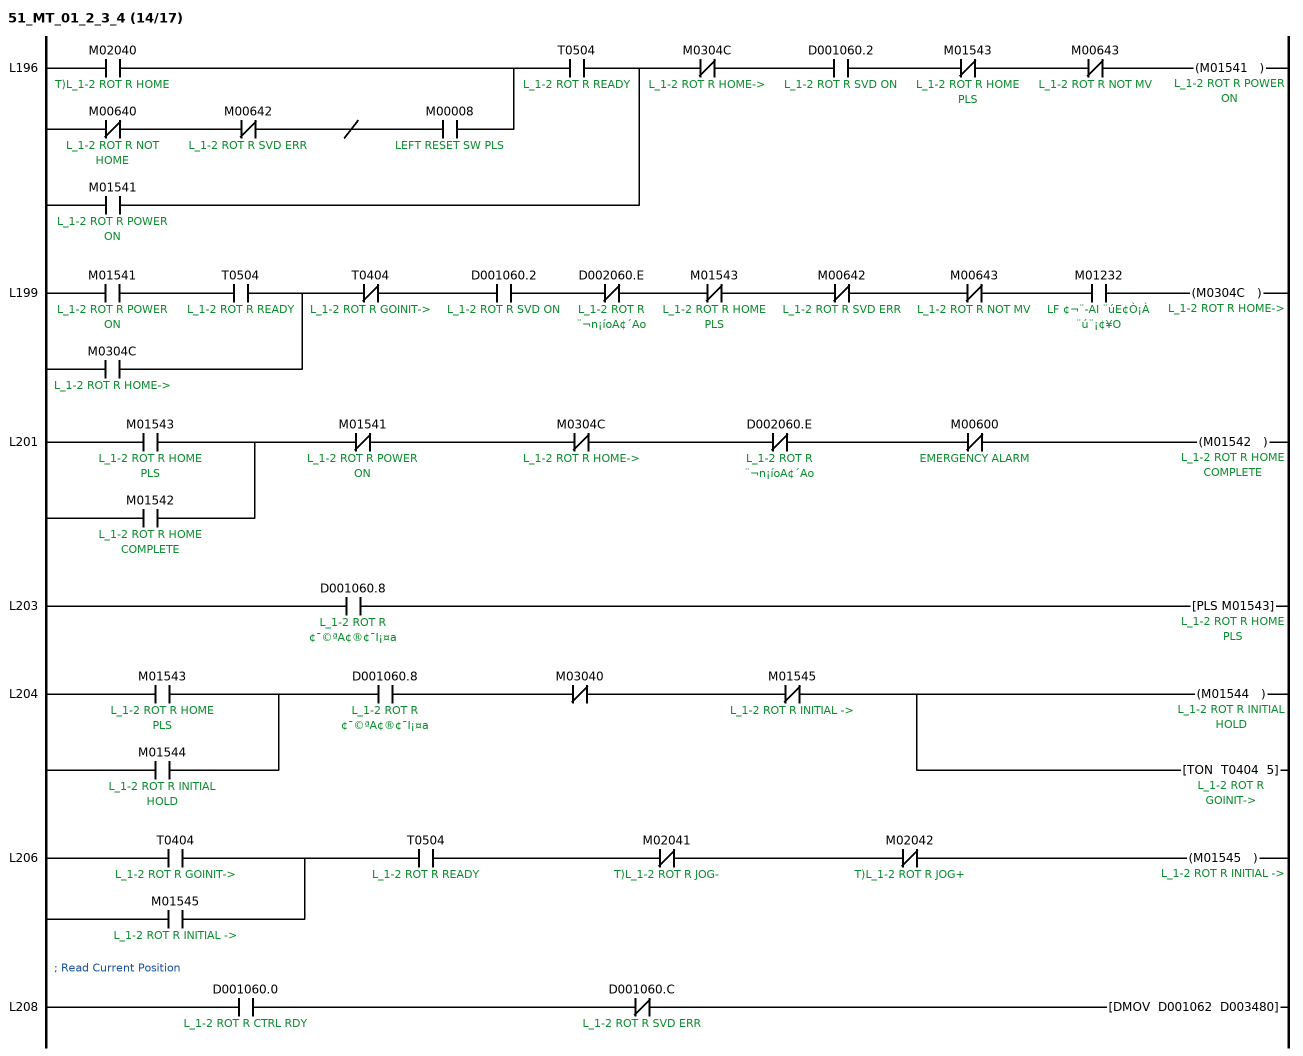
; L196
LOAD      M02040	// T)L_1-2 ROT R HOME
LOAD NOT  M00640	// L_1-2 ROT R NOT HOME
AND NOT   M00642	// L_1-2 ROT R SVD ERR
NOT
AND       M00008	// LEFT RESET SW PLS
OR LOAD
AND       T0504	// L_1-2 ROT R READY
OR        M01541	// L_1-2 ROT R POWER ON
AND NOT   M0304C	// L_1-2 ROT R HOME->
AND       D001060.2	// L_1-2 ROT R SVD ON
AND NOT   M01543	// L_1-2 ROT R HOME PLS
AND NOT   M00643	// L_1-2 ROT R NOT MV
OUT       M01541	// L_1-2 ROT R POWER ON
; L199
LOAD      M01541	// L_1-2 ROT R POWER ON
AND       T0504	// L_1-2 ROT R READY
OR        M0304C	// L_1-2 ROT R HOME->
AND NOT   T0404	// L_1-2 ROT R GOINIT->
AND       D001060.2	// L_1-2 ROT R SVD ON
AND NOT   D002060.E	// L_1-2 ROT R ¨¬n¡íoA¢´Ao
AND NOT   M01543	// L_1-2 ROT R HOME PLS
AND NOT   M00642	// L_1-2 ROT R SVD ERR
AND NOT   M00643	// L_1-2 ROT R NOT MV
AND       M01232	// LF ¢¬¨­AI ¨úE¢Ò¡À ¨ú¨¡¢¥O
OUT       M0304C	// L_1-2 ROT R HOME->
; L201
LOAD      M01543	// L_1-2 ROT R HOME PLS
OR        M01542	// L_1-2 ROT R HOME COMPLETE
AND NOT   M01541	// L_1-2 ROT R POWER ON
AND NOT   M0304C	// L_1-2 ROT R HOME->
AND NOT   D002060.E	// L_1-2 ROT R ¨¬n¡íoA¢´Ao
AND NOT   M00600	// EMERGENCY ALARM
OUT       M01542	// L_1-2 ROT R HOME COMPLETE
; L203
LOAD      D001060.8	// L_1-2 ROT R ¢¯©ªA¢®¢¯I¡¤a
OUTP      M01543	// L_1-2 ROT R HOME PLS
; L204
LOAD      M01543	// L_1-2 ROT R HOME PLS
OR        M01544	// L_1-2 ROT R INITIAL HOLD
AND       D001060.8	// L_1-2 ROT R ¢¯©ªA¢®¢¯I¡¤a
AND NOT   M03040
AND NOT   M01545	// L_1-2 ROT R INITIAL ->
OUT       M01544	// L_1-2 ROT R INITIAL HOLD
TON       T0404 5	// L_1-2 ROT R GOINIT->
; L206
LOAD      T0404	// L_1-2 ROT R GOINIT->
OR        M01545	// L_1-2 ROT R INITIAL ->
AND       T0504	// L_1-2 ROT R READY
AND NOT   M02041	// T)L_1-2 ROT R JOG-
AND NOT   M02042	// T)L_1-2 ROT R JOG+
OUT       M01545	// L_1-2 ROT R INITIAL ->
; L208
LOAD      D001060.0	// L_1-2 ROT R CTRL RDY
AND NOT   D001060.C	// L_1-2 ROT R SVD ERR
DMOV      D001062 D003480
// output comment: Read Current Position

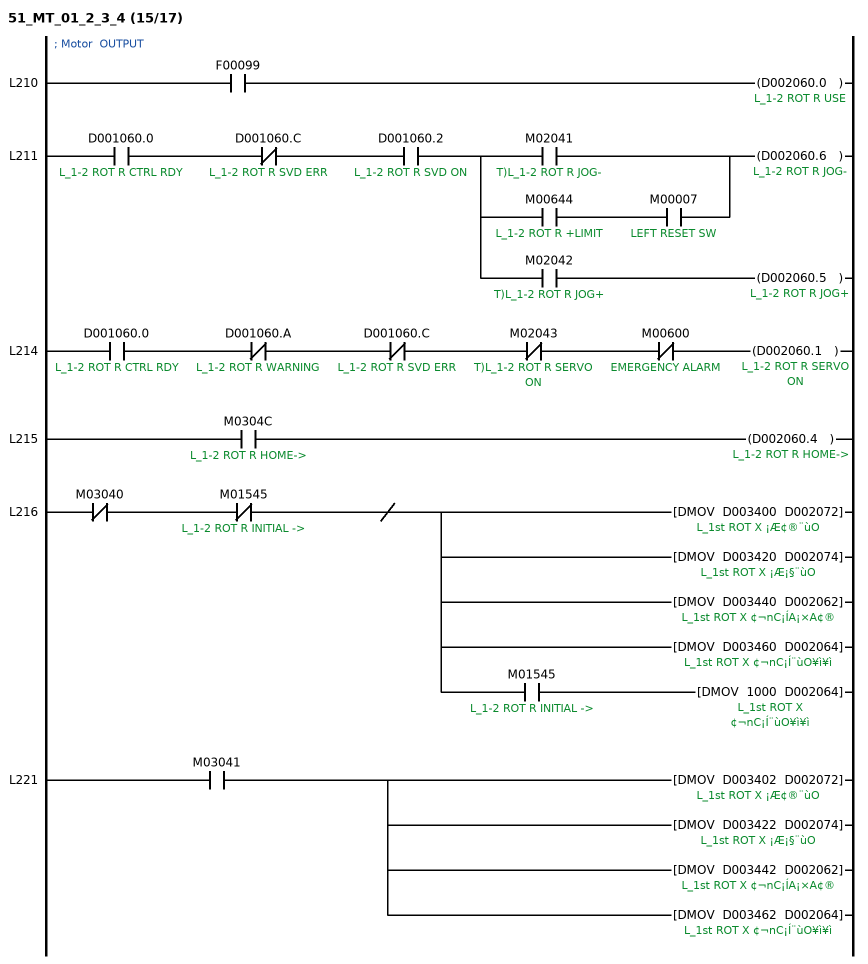
//  Motor  OUTPUT
; L210
LOAD      F00099
OUT       D002060.0	// L_1-2 ROT R USE
; L211
LOAD      D001060.0	// L_1-2 ROT R CTRL RDY
AND NOT   D001060.C	// L_1-2 ROT R SVD ERR
AND       D001060.2	// L_1-2 ROT R SVD ON
MPUSH
LOAD      M02041	// T)L_1-2 ROT R JOG-
LOAD      M00644	// L_1-2 ROT R +LIMIT
AND       M00007	// LEFT RESET SW
OR LOAD
AND LOAD
OUT       D002060.6	// L_1-2 ROT R JOG-
MPOP
AND       M02042	// T)L_1-2 ROT R JOG+
OUT       D002060.5	// L_1-2 ROT R JOG+
; L214
LOAD      D001060.0	// L_1-2 ROT R CTRL RDY
AND NOT   D001060.A	// L_1-2 ROT R WARNING
AND NOT   D001060.C	// L_1-2 ROT R SVD ERR
AND NOT   M02043	// T)L_1-2 ROT R SERVO ON
AND NOT   M00600	// EMERGENCY ALARM
OUT       D002060.1	// L_1-2 ROT R SERVO ON
; L215
LOAD      M0304C	// L_1-2 ROT R HOME->
OUT       D002060.4	// L_1-2 ROT R HOME->
; L216
LOAD NOT  M03040
AND NOT   M01545	// L_1-2 ROT R INITIAL ->
NOT
DMOV      D003400 D002072	// L_1st ROT X ¡Æ¢®¨ùO
DMOV      D003420 D002074	// L_1st ROT X ¡Æ¡§¨ùO
DMOV      D003440 D002062	// L_1st ROT X ¢¬nC¡ÍA¡×A¢®
DMOV      D003460 D002064	// L_1st ROT X ¢¬nC¡Í¨ùO¥ì¥ì
AND       M01545	// L_1-2 ROT R INITIAL ->
DMOV      1000 D002064	// L_1st ROT X ¢¬nC¡Í¨ùO¥ì¥ì
; L221
LOAD      M03041
DMOV      D003402 D002072	// L_1st ROT X ¡Æ¢®¨ùO
DMOV      D003422 D002074	// L_1st ROT X ¡Æ¡§¨ùO
DMOV      D003442 D002062	// L_1st ROT X ¢¬nC¡ÍA¡×A¢®
DMOV      D003462 D002064	// L_1st ROT X ¢¬nC¡Í¨ùO¥ì¥ì

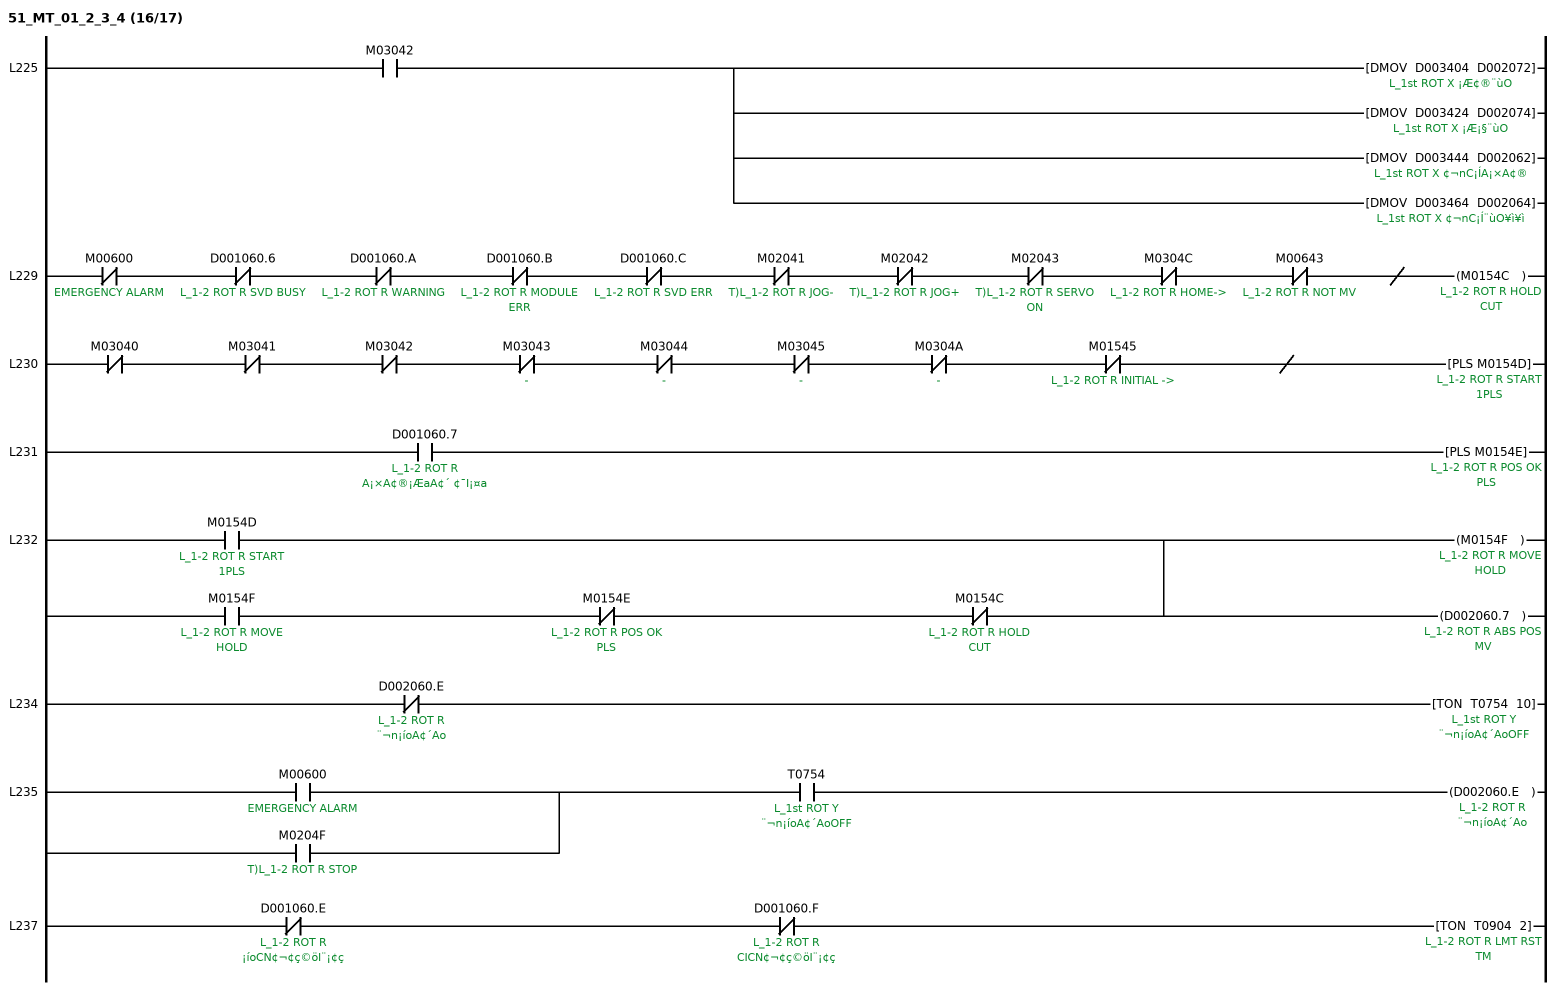
; L225
LOAD      M03042
DMOV      D003404 D002072	// L_1st ROT X ¡Æ¢®¨ùO
DMOV      D003424 D002074	// L_1st ROT X ¡Æ¡§¨ùO
DMOV      D003444 D002062	// L_1st ROT X ¢¬nC¡ÍA¡×A¢®
DMOV      D003464 D002064	// L_1st ROT X ¢¬nC¡Í¨ùO¥ì¥ì
; L229
LOAD NOT  M00600	// EMERGENCY ALARM
AND NOT   D001060.6	// L_1-2 ROT R SVD BUSY
AND NOT   D001060.A	// L_1-2 ROT R WARNING
AND NOT   D001060.B	// L_1-2 ROT R MODULE ERR
AND NOT   D001060.C	// L_1-2 ROT R SVD ERR
AND NOT   M02041	// T)L_1-2 ROT R JOG-
AND NOT   M02042	// T)L_1-2 ROT R JOG+
AND NOT   M02043	// T)L_1-2 ROT R SERVO ON
AND NOT   M0304C	// L_1-2 ROT R HOME->
AND NOT   M00643	// L_1-2 ROT R NOT MV
NOT
OUT       M0154C	// L_1-2 ROT R HOLD CUT
; L230
LOAD NOT  M03040
AND NOT   M03041
AND NOT   M03042
AND NOT   M03043	// -
AND NOT   M03044	// -
AND NOT   M03045	// -
AND NOT   M0304A	// -
AND NOT   M01545	// L_1-2 ROT R INITIAL ->
NOT
OUTP      M0154D	// L_1-2 ROT R START 1PLS
; L231
LOAD      D001060.7	// L_1-2 ROT R A¡×A¢®¡ÆaA¢´ ¢¯I¡¤a
OUTP      M0154E	// L_1-2 ROT R POS OK PLS
; L232
LOAD      M0154D	// L_1-2 ROT R START 1PLS
LOAD      M0154F	// L_1-2 ROT R MOVE HOLD
AND NOT   M0154E	// L_1-2 ROT R POS OK PLS
AND NOT   M0154C	// L_1-2 ROT R HOLD CUT
OR LOAD
OUT       M0154F	// L_1-2 ROT R MOVE HOLD
OUT       D002060.7	// L_1-2 ROT R ABS POS MV
; L234
LOAD NOT  D002060.E	// L_1-2 ROT R ¨¬n¡íoA¢´Ao
TON       T0754 10	// L_1st ROT Y ¨¬n¡íoA¢´AoOFF
; L235
LOAD      M00600	// EMERGENCY ALARM
OR        M0204F	// T)L_1-2 ROT R STOP
AND       T0754	// L_1st ROT Y ¨¬n¡íoA¢´AoOFF
OUT       D002060.E	// L_1-2 ROT R ¨¬n¡íoA¢´Ao
; L237
LOAD NOT  D001060.E	// L_1-2 ROT R ¡íoCN¢¬¢ç©öI¨¡¢ç
AND NOT   D001060.F	// L_1-2 ROT R CICN¢¬¢ç©öI¨¡¢ç
TON       T0904 2	// L_1-2 ROT R LMT RST TM

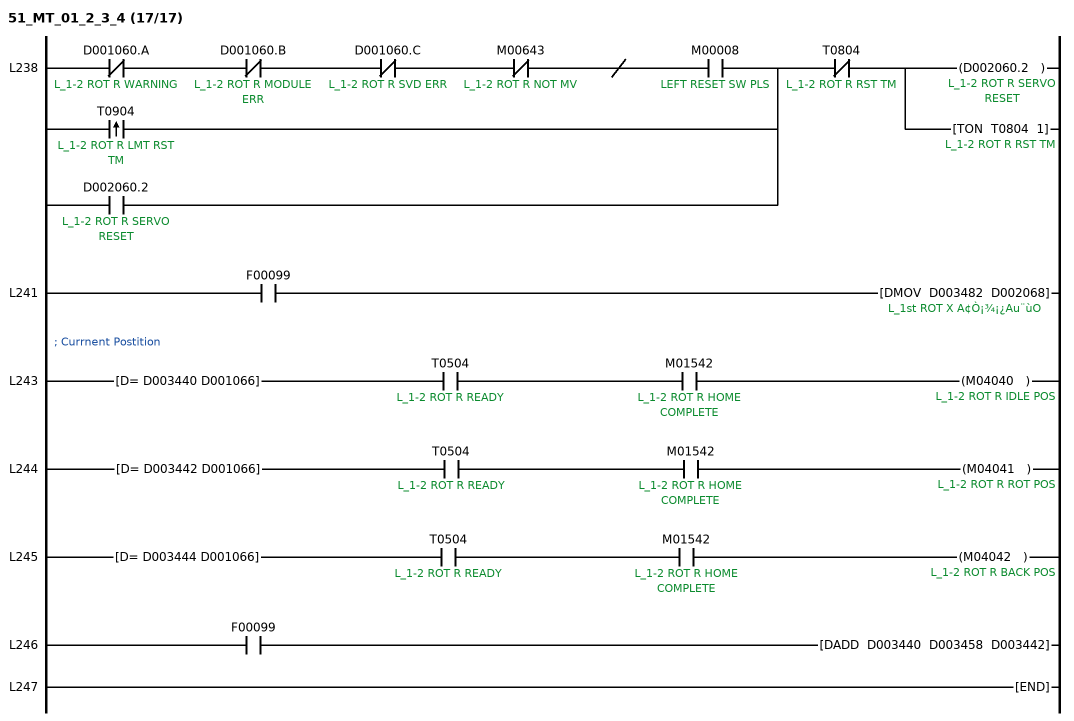
; L238
LOAD NOT  D001060.A	// L_1-2 ROT R WARNING
AND NOT   D001060.B	// L_1-2 ROT R MODULE ERR
AND NOT   D001060.C	// L_1-2 ROT R SVD ERR
AND NOT   M00643	// L_1-2 ROT R NOT MV
NOT
AND       M00008	// LEFT RESET SW PLS
ORP       T0904	// L_1-2 ROT R LMT RST TM
OR        D002060.2	// L_1-2 ROT R SERVO RESET
AND NOT   T0804	// L_1-2 ROT R RST TM
OUT       D002060.2	// L_1-2 ROT R SERVO RESET
TON       T0804 1	// L_1-2 ROT R RST TM
; L241
LOAD      F00099
DMOV      D003482 D002068	// L_1st ROT X A¢Ò¡¾¡¿Au¨ùO
// Currnent Postition
; L243
LOADD=    D003440 D001066
AND       T0504	// L_1-2 ROT R READY
AND       M01542	// L_1-2 ROT R HOME COMPLETE
OUT       M04040	// L_1-2 ROT R IDLE POS
; L244
LOADD=    D003442 D001066
AND       T0504	// L_1-2 ROT R READY
AND       M01542	// L_1-2 ROT R HOME COMPLETE
OUT       M04041	// L_1-2 ROT R ROT POS
; L245
LOADD=    D003444 D001066
AND       T0504	// L_1-2 ROT R READY
AND       M01542	// L_1-2 ROT R HOME COMPLETE
OUT       M04042	// L_1-2 ROT R BACK POS
; L246
LOAD      F00099
DADD      D003440 D003458 D003442
; L247
END

PROGRAM 52_MT_05_6_7_8 (task: ¨ö¨¬A¥ì CA¡¤I¡¾¡¿¡¤¡Í)

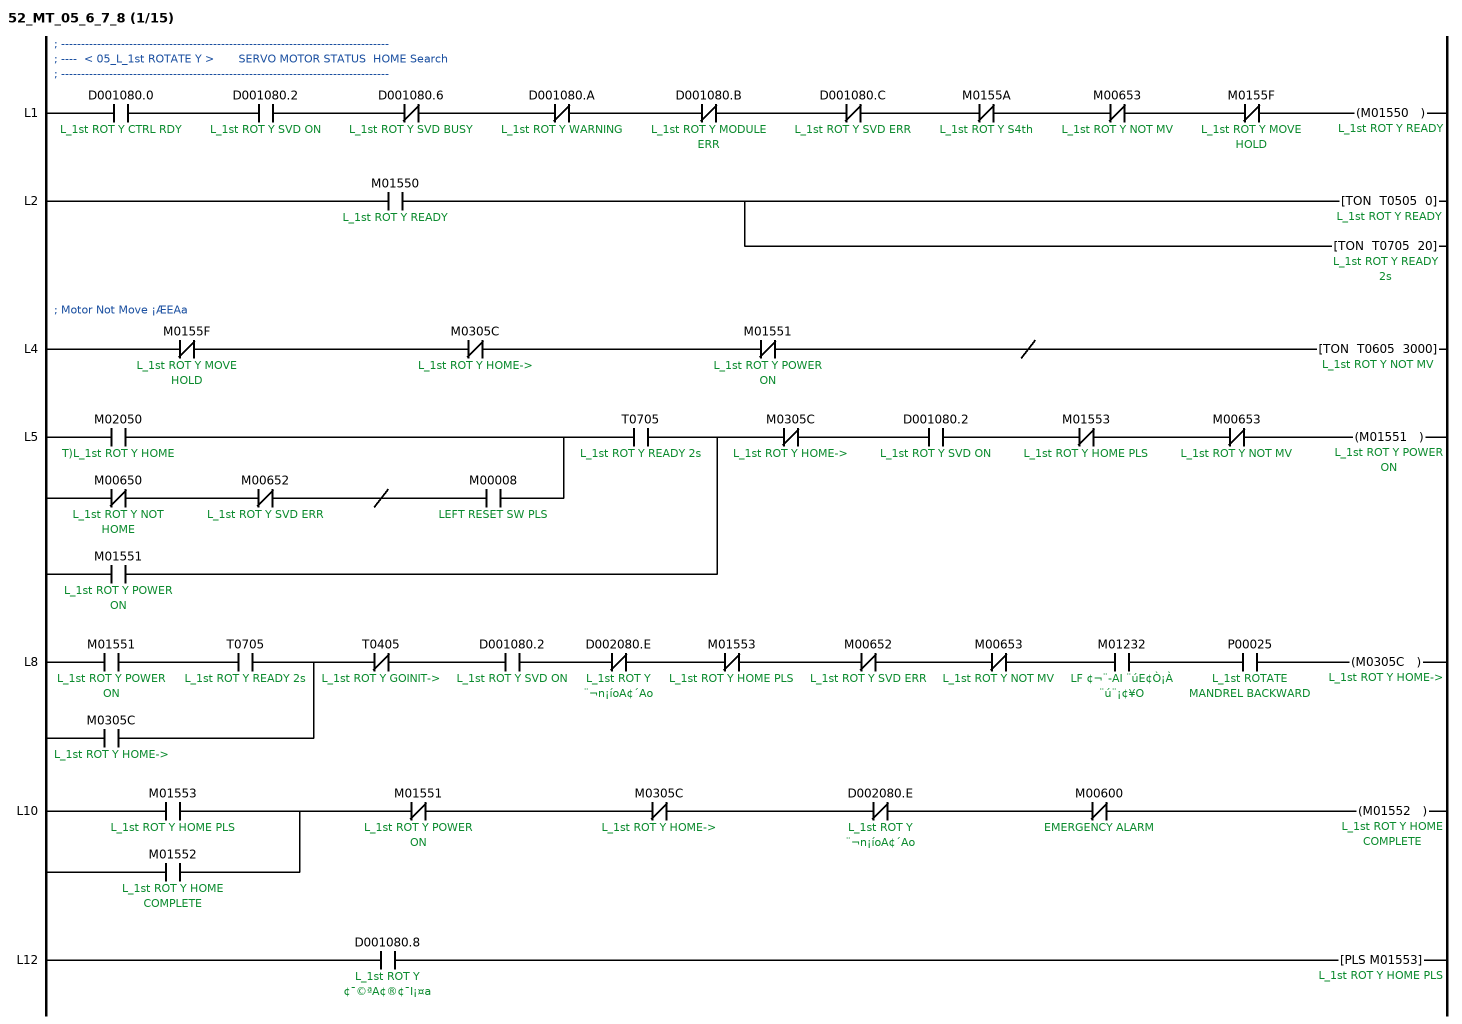
// ----------------------------------------------------------------------------------
// 
// ----  < 05_L_1st ROTATE Y >       SERVO MOTOR STATUS  HOME Search
// 
// ----------------------------------------------------------------------------------
; L1
LOAD      D001080.0	// L_1st ROT Y CTRL RDY
AND       D001080.2	// L_1st ROT Y SVD ON
AND NOT   D001080.6	// L_1st ROT Y SVD BUSY
AND NOT   D001080.A	// L_1st ROT Y WARNING
AND NOT   D001080.B	// L_1st ROT Y MODULE ERR
AND NOT   D001080.C	// L_1st ROT Y SVD ERR
AND NOT   M0155A	// L_1st ROT Y S4th
AND NOT   M00653	// L_1st ROT Y NOT MV
AND NOT   M0155F	// L_1st ROT Y MOVE HOLD
OUT       M01550	// L_1st ROT Y READY
; L2
LOAD      M01550	// L_1st ROT Y READY
TON       T0505 0	// L_1st ROT Y READY
TON       T0705 20	// L_1st ROT Y READY 2s
; L4
LOAD NOT  M0155F	// L_1st ROT Y MOVE HOLD
AND NOT   M0305C	// L_1st ROT Y HOME->
AND NOT   M01551	// L_1st ROT Y POWER ON
NOT
TON       T0605 3000	// L_1st ROT Y NOT MV
// output comment: Motor Not Move ¡ÆEAa
; L5
LOAD      M02050	// T)L_1st ROT Y HOME
LOAD NOT  M00650	// L_1st ROT Y NOT HOME
AND NOT   M00652	// L_1st ROT Y SVD ERR
NOT
AND       M00008	// LEFT RESET SW PLS
OR LOAD
AND       T0705	// L_1st ROT Y READY 2s
OR        M01551	// L_1st ROT Y POWER ON
AND NOT   M0305C	// L_1st ROT Y HOME->
AND       D001080.2	// L_1st ROT Y SVD ON
AND NOT   M01553	// L_1st ROT Y HOME PLS
AND NOT   M00653	// L_1st ROT Y NOT MV
OUT       M01551	// L_1st ROT Y POWER ON
; L8
LOAD      M01551	// L_1st ROT Y POWER ON
AND       T0705	// L_1st ROT Y READY 2s
OR        M0305C	// L_1st ROT Y HOME->
AND NOT   T0405	// L_1st ROT Y GOINIT->
AND       D001080.2	// L_1st ROT Y SVD ON
AND NOT   D002080.E	// L_1st ROT Y ¨¬n¡íoA¢´Ao
AND NOT   M01553	// L_1st ROT Y HOME PLS
AND NOT   M00652	// L_1st ROT Y SVD ERR
AND NOT   M00653	// L_1st ROT Y NOT MV
AND       M01232	// LF ¢¬¨­AI ¨úE¢Ò¡À ¨ú¨¡¢¥O
AND       P00025	// L_1st ROTATE MANDREL BACKWARD
OUT       M0305C	// L_1st ROT Y HOME->
; L10
LOAD      M01553	// L_1st ROT Y HOME PLS
OR        M01552	// L_1st ROT Y HOME COMPLETE
AND NOT   M01551	// L_1st ROT Y POWER ON
AND NOT   M0305C	// L_1st ROT Y HOME->
AND NOT   D002080.E	// L_1st ROT Y ¨¬n¡íoA¢´Ao
AND NOT   M00600	// EMERGENCY ALARM
OUT       M01552	// L_1st ROT Y HOME COMPLETE
; L12
LOAD      D001080.8	// L_1st ROT Y ¢¯©ªA¢®¢¯I¡¤a
OUTP      M01553	// L_1st ROT Y HOME PLS

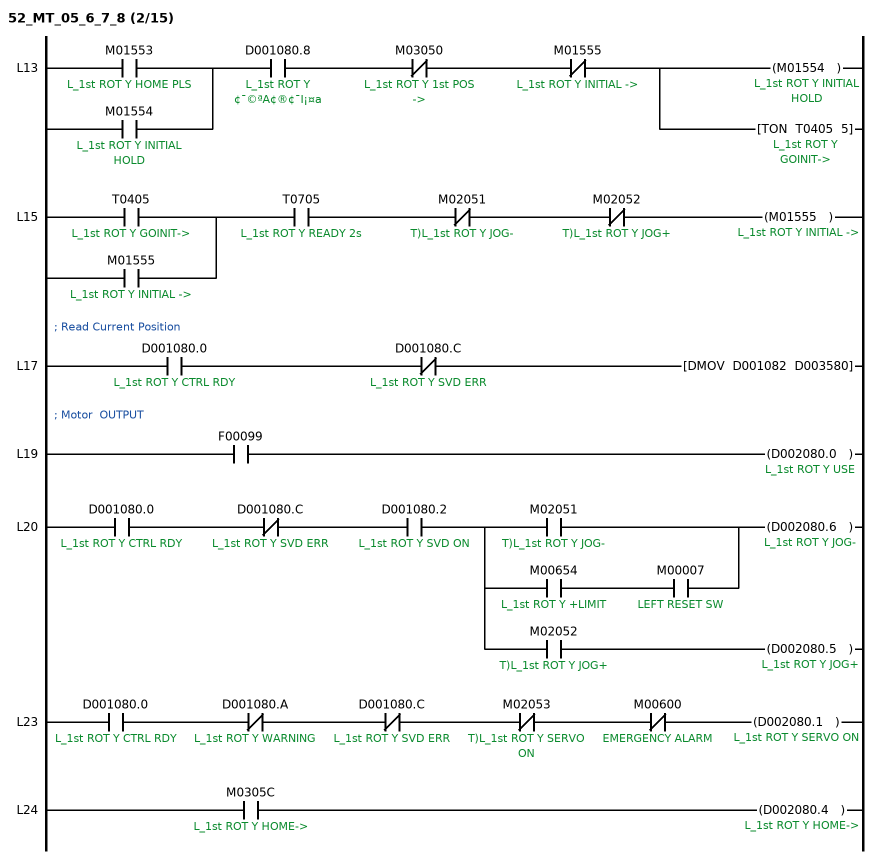
; L13
LOAD      M01553	// L_1st ROT Y HOME PLS
OR        M01554	// L_1st ROT Y INITIAL HOLD
AND       D001080.8	// L_1st ROT Y ¢¯©ªA¢®¢¯I¡¤a
AND NOT   M03050	// L_1st ROT Y 1st POS ->
AND NOT   M01555	// L_1st ROT Y INITIAL ->
OUT       M01554	// L_1st ROT Y INITIAL HOLD
TON       T0405 5	// L_1st ROT Y GOINIT->
; L15
LOAD      T0405	// L_1st ROT Y GOINIT->
OR        M01555	// L_1st ROT Y INITIAL ->
AND       T0705	// L_1st ROT Y READY 2s
AND NOT   M02051	// T)L_1st ROT Y JOG-
AND NOT   M02052	// T)L_1st ROT Y JOG+
OUT       M01555	// L_1st ROT Y INITIAL ->
; L17
LOAD      D001080.0	// L_1st ROT Y CTRL RDY
AND NOT   D001080.C	// L_1st ROT Y SVD ERR
DMOV      D001082 D003580
// output comment: Read Current Position
//  Motor  OUTPUT
; L19
LOAD      F00099
OUT       D002080.0	// L_1st ROT Y USE
; L20
LOAD      D001080.0	// L_1st ROT Y CTRL RDY
AND NOT   D001080.C	// L_1st ROT Y SVD ERR
AND       D001080.2	// L_1st ROT Y SVD ON
MPUSH
LOAD      M02051	// T)L_1st ROT Y JOG-
LOAD      M00654	// L_1st ROT Y +LIMIT
AND       M00007	// LEFT RESET SW
OR LOAD
AND LOAD
OUT       D002080.6	// L_1st ROT Y JOG-
MPOP
AND       M02052	// T)L_1st ROT Y JOG+
OUT       D002080.5	// L_1st ROT Y JOG+
; L23
LOAD      D001080.0	// L_1st ROT Y CTRL RDY
AND NOT   D001080.A	// L_1st ROT Y WARNING
AND NOT   D001080.C	// L_1st ROT Y SVD ERR
AND NOT   M02053	// T)L_1st ROT Y SERVO ON
AND NOT   M00600	// EMERGENCY ALARM
OUT       D002080.1	// L_1st ROT Y SERVO ON
; L24
LOAD      M0305C	// L_1st ROT Y HOME->
OUT       D002080.4	// L_1st ROT Y HOME->

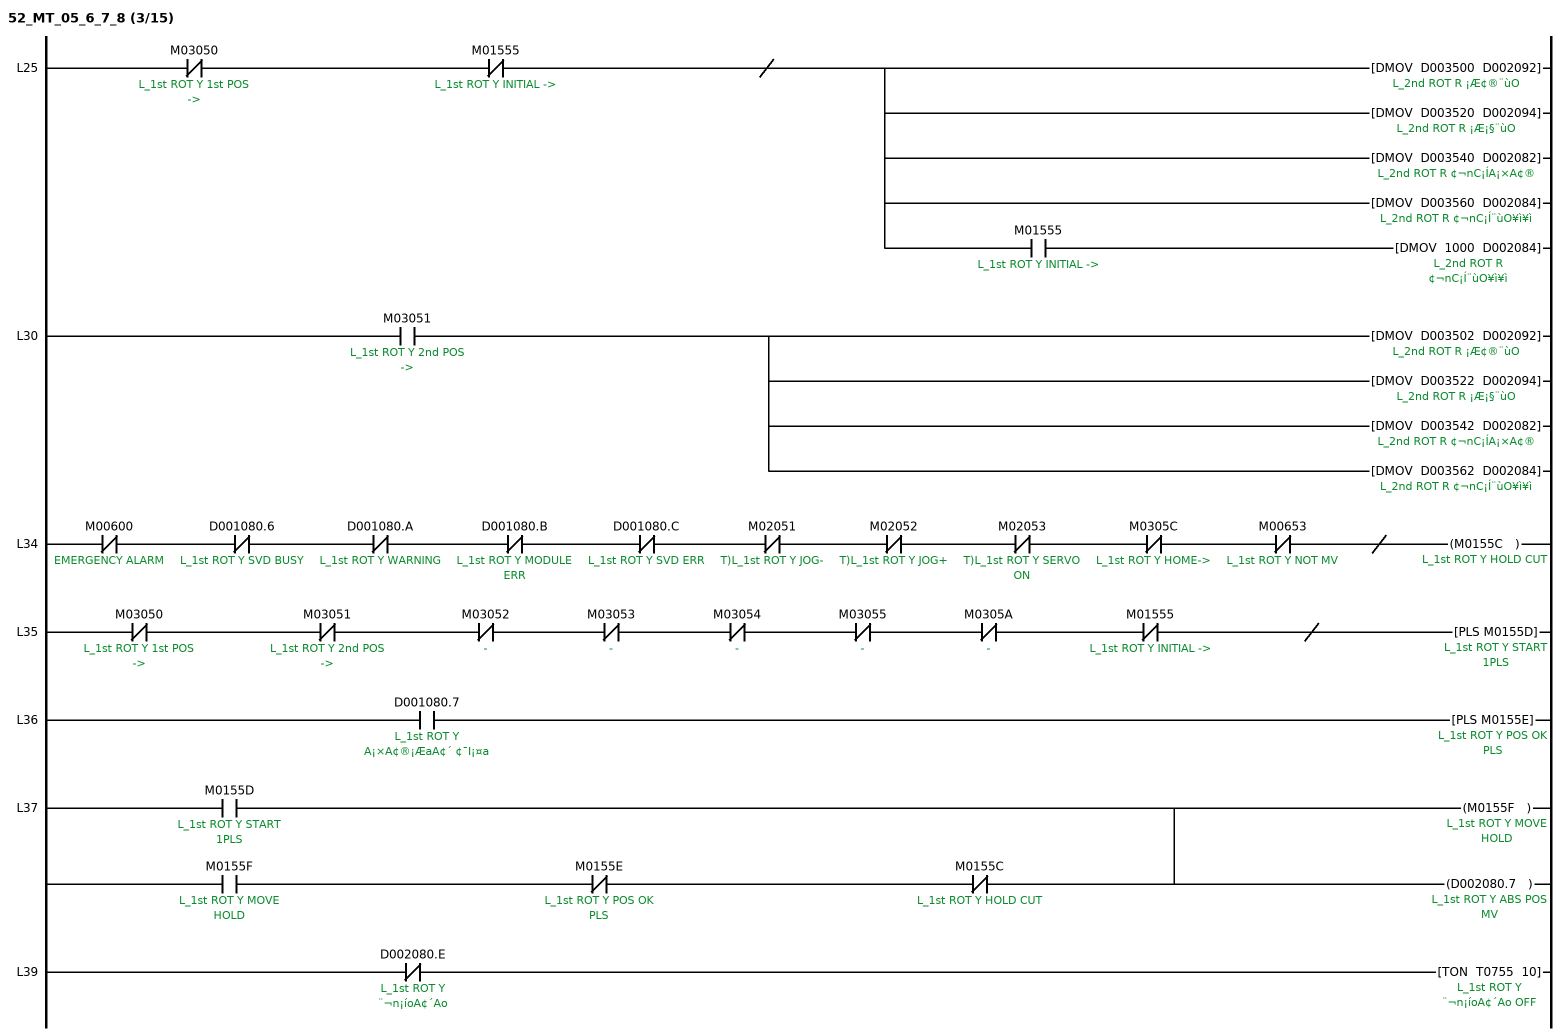
; L25
LOAD NOT  M03050	// L_1st ROT Y 1st POS ->
AND NOT   M01555	// L_1st ROT Y INITIAL ->
NOT
DMOV      D003500 D002092	// L_2nd ROT R ¡Æ¢®¨ùO
DMOV      D003520 D002094	// L_2nd ROT R ¡Æ¡§¨ùO
DMOV      D003540 D002082	// L_2nd ROT R ¢¬nC¡ÍA¡×A¢®
DMOV      D003560 D002084	// L_2nd ROT R ¢¬nC¡Í¨ùO¥ì¥ì
AND       M01555	// L_1st ROT Y INITIAL ->
DMOV      1000 D002084	// L_2nd ROT R ¢¬nC¡Í¨ùO¥ì¥ì
; L30
LOAD      M03051	// L_1st ROT Y 2nd POS ->
DMOV      D003502 D002092	// L_2nd ROT R ¡Æ¢®¨ùO
DMOV      D003522 D002094	// L_2nd ROT R ¡Æ¡§¨ùO
DMOV      D003542 D002082	// L_2nd ROT R ¢¬nC¡ÍA¡×A¢®
DMOV      D003562 D002084	// L_2nd ROT R ¢¬nC¡Í¨ùO¥ì¥ì
; L34
LOAD NOT  M00600	// EMERGENCY ALARM
AND NOT   D001080.6	// L_1st ROT Y SVD BUSY
AND NOT   D001080.A	// L_1st ROT Y WARNING
AND NOT   D001080.B	// L_1st ROT Y MODULE ERR
AND NOT   D001080.C	// L_1st ROT Y SVD ERR
AND NOT   M02051	// T)L_1st ROT Y JOG-
AND NOT   M02052	// T)L_1st ROT Y JOG+
AND NOT   M02053	// T)L_1st ROT Y SERVO ON
AND NOT   M0305C	// L_1st ROT Y HOME->
AND NOT   M00653	// L_1st ROT Y NOT MV
NOT
OUT       M0155C	// L_1st ROT Y HOLD CUT
; L35
LOAD NOT  M03050	// L_1st ROT Y 1st POS ->
AND NOT   M03051	// L_1st ROT Y 2nd POS ->
AND NOT   M03052	// -
AND NOT   M03053	// -
AND NOT   M03054	// -
AND NOT   M03055	// -
AND NOT   M0305A	// -
AND NOT   M01555	// L_1st ROT Y INITIAL ->
NOT
OUTP      M0155D	// L_1st ROT Y START 1PLS
; L36
LOAD      D001080.7	// L_1st ROT Y A¡×A¢®¡ÆaA¢´ ¢¯I¡¤a
OUTP      M0155E	// L_1st ROT Y POS OK PLS
; L37
LOAD      M0155D	// L_1st ROT Y START 1PLS
LOAD      M0155F	// L_1st ROT Y MOVE HOLD
AND NOT   M0155E	// L_1st ROT Y POS OK PLS
AND NOT   M0155C	// L_1st ROT Y HOLD CUT
OR LOAD
OUT       M0155F	// L_1st ROT Y MOVE HOLD
OUT       D002080.7	// L_1st ROT Y ABS POS MV
; L39
LOAD NOT  D002080.E	// L_1st ROT Y ¨¬n¡íoA¢´Ao
TON       T0755 10	// L_1st ROT Y ¨¬n¡íoA¢´Ao OFF

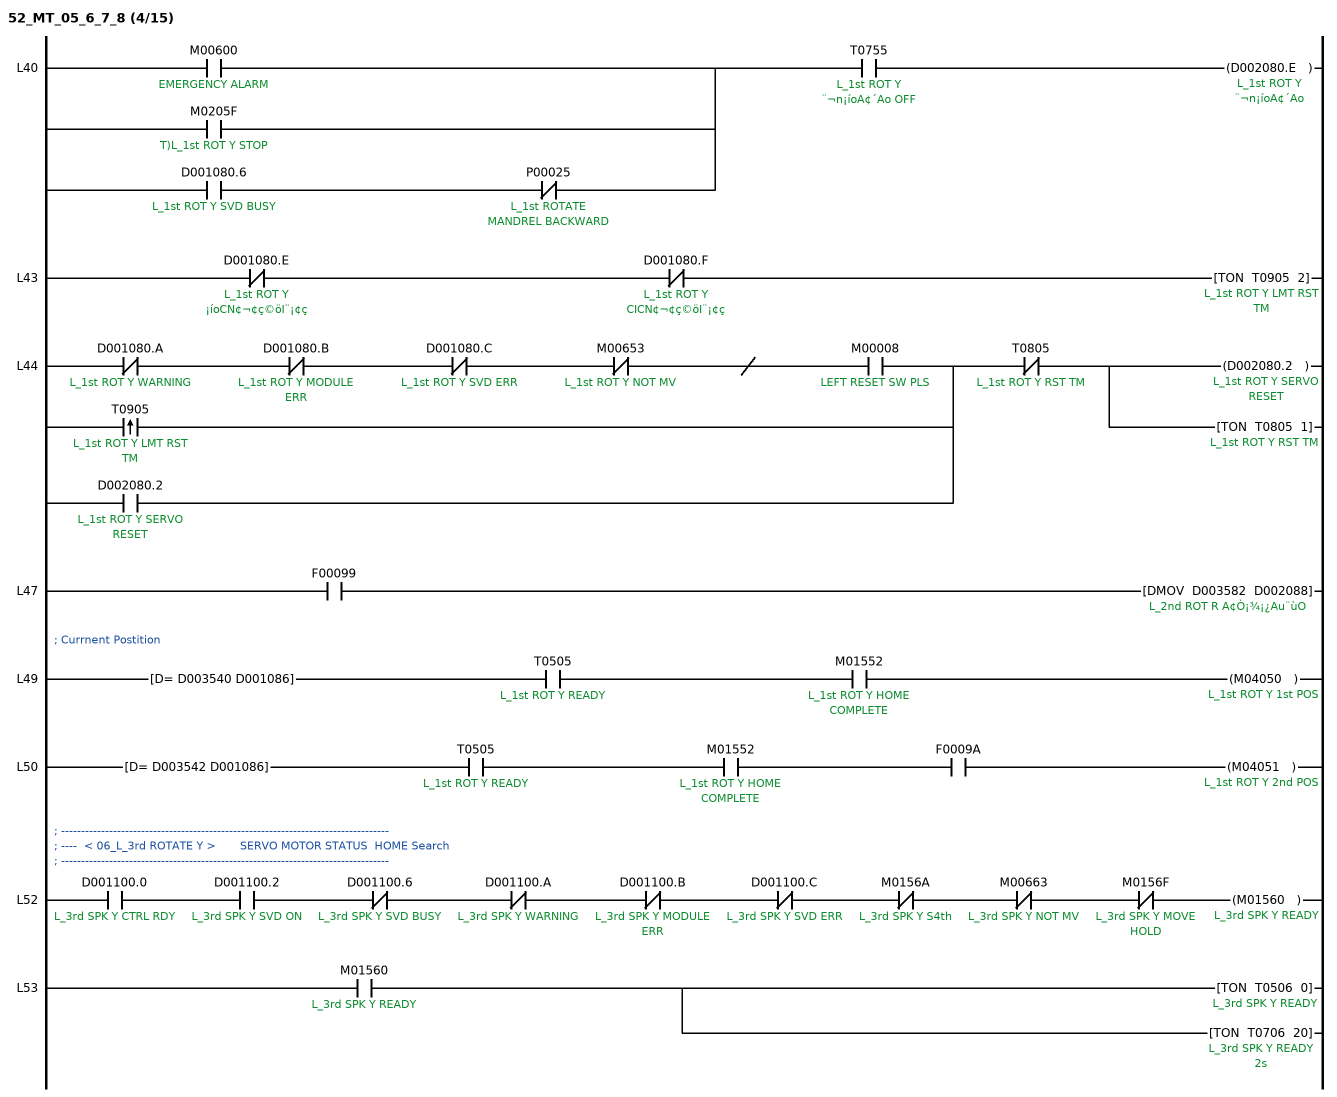
; L40
LOAD      M00600	// EMERGENCY ALARM
OR        M0205F	// T)L_1st ROT Y STOP
LOAD      D001080.6	// L_1st ROT Y SVD BUSY
AND NOT   P00025	// L_1st ROTATE MANDREL BACKWARD
OR LOAD
AND       T0755	// L_1st ROT Y ¨¬n¡íoA¢´Ao OFF
OUT       D002080.E	// L_1st ROT Y ¨¬n¡íoA¢´Ao
; L43
LOAD NOT  D001080.E	// L_1st ROT Y ¡íoCN¢¬¢ç©öI¨¡¢ç
AND NOT   D001080.F	// L_1st ROT Y CICN¢¬¢ç©öI¨¡¢ç
TON       T0905 2	// L_1st ROT Y LMT RST TM
; L44
LOAD NOT  D001080.A	// L_1st ROT Y WARNING
AND NOT   D001080.B	// L_1st ROT Y MODULE ERR
AND NOT   D001080.C	// L_1st ROT Y SVD ERR
AND NOT   M00653	// L_1st ROT Y NOT MV
NOT
AND       M00008	// LEFT RESET SW PLS
ORP       T0905	// L_1st ROT Y LMT RST TM
OR        D002080.2	// L_1st ROT Y SERVO RESET
AND NOT   T0805	// L_1st ROT Y RST TM
OUT       D002080.2	// L_1st ROT Y SERVO RESET
TON       T0805 1	// L_1st ROT Y RST TM
; L47
LOAD      F00099
DMOV      D003582 D002088	// L_2nd ROT R A¢Ò¡¾¡¿Au¨ùO
// Currnent Postition
; L49
LOADD=    D003540 D001086
AND       T0505	// L_1st ROT Y READY
AND       M01552	// L_1st ROT Y HOME COMPLETE
OUT       M04050	// L_1st ROT Y 1st POS
; L50
LOADD=    D003542 D001086
AND       T0505	// L_1st ROT Y READY
AND       M01552	// L_1st ROT Y HOME COMPLETE
AND       F0009A
OUT       M04051	// L_1st ROT Y 2nd POS
// ----------------------------------------------------------------------------------
// 
// ----  < 06_L_3rd ROTATE Y >       SERVO MOTOR STATUS  HOME Search
// 
// ----------------------------------------------------------------------------------
; L52
LOAD      D001100.0	// L_3rd SPK Y CTRL RDY
AND       D001100.2	// L_3rd SPK Y SVD ON
AND NOT   D001100.6	// L_3rd SPK Y SVD BUSY
AND NOT   D001100.A	// L_3rd SPK Y WARNING
AND NOT   D001100.B	// L_3rd SPK Y MODULE ERR
AND NOT   D001100.C	// L_3rd SPK Y SVD ERR
AND NOT   M0156A	// L_3rd SPK Y S4th
AND NOT   M00663	// L_3rd SPK Y NOT MV
AND NOT   M0156F	// L_3rd SPK Y MOVE HOLD
OUT       M01560	// L_3rd SPK Y READY
; L53
LOAD      M01560	// L_3rd SPK Y READY
TON       T0506 0	// L_3rd SPK Y READY
TON       T0706 20	// L_3rd SPK Y READY 2s

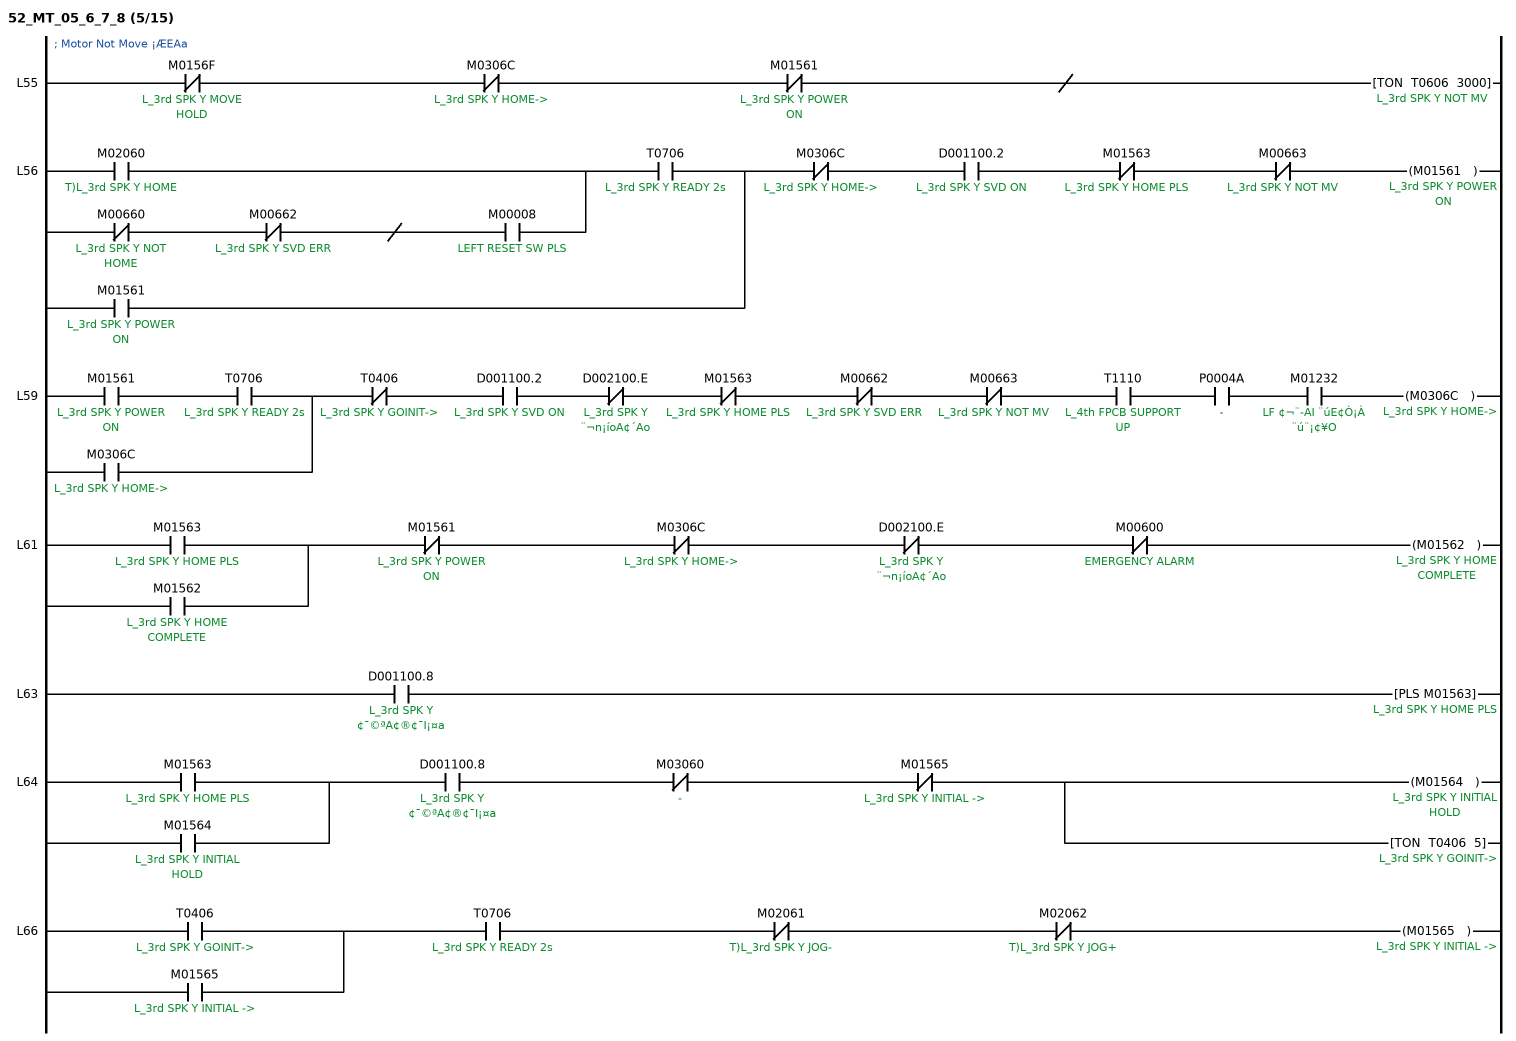
; L55
LOAD NOT  M0156F	// L_3rd SPK Y MOVE HOLD
AND NOT   M0306C	// L_3rd SPK Y HOME->
AND NOT   M01561	// L_3rd SPK Y POWER ON
NOT
TON       T0606 3000	// L_3rd SPK Y NOT MV
// output comment: Motor Not Move ¡ÆEAa
; L56
LOAD      M02060	// T)L_3rd SPK Y HOME
LOAD NOT  M00660	// L_3rd SPK Y NOT HOME
AND NOT   M00662	// L_3rd SPK Y SVD ERR
NOT
AND       M00008	// LEFT RESET SW PLS
OR LOAD
AND       T0706	// L_3rd SPK Y READY 2s
OR        M01561	// L_3rd SPK Y POWER ON
AND NOT   M0306C	// L_3rd SPK Y HOME->
AND       D001100.2	// L_3rd SPK Y SVD ON
AND NOT   M01563	// L_3rd SPK Y HOME PLS
AND NOT   M00663	// L_3rd SPK Y NOT MV
OUT       M01561	// L_3rd SPK Y POWER ON
; L59
LOAD      M01561	// L_3rd SPK Y POWER ON
AND       T0706	// L_3rd SPK Y READY 2s
OR        M0306C	// L_3rd SPK Y HOME->
AND NOT   T0406	// L_3rd SPK Y GOINIT->
AND       D001100.2	// L_3rd SPK Y SVD ON
AND NOT   D002100.E	// L_3rd SPK Y ¨¬n¡íoA¢´Ao
AND NOT   M01563	// L_3rd SPK Y HOME PLS
AND NOT   M00662	// L_3rd SPK Y SVD ERR
AND NOT   M00663	// L_3rd SPK Y NOT MV
AND       T1110	// L_4th FPCB SUPPORT UP
AND       P0004A	// -
AND       M01232	// LF ¢¬¨­AI ¨úE¢Ò¡À ¨ú¨¡¢¥O
OUT       M0306C	// L_3rd SPK Y HOME->
; L61
LOAD      M01563	// L_3rd SPK Y HOME PLS
OR        M01562	// L_3rd SPK Y HOME COMPLETE
AND NOT   M01561	// L_3rd SPK Y POWER ON
AND NOT   M0306C	// L_3rd SPK Y HOME->
AND NOT   D002100.E	// L_3rd SPK Y ¨¬n¡íoA¢´Ao
AND NOT   M00600	// EMERGENCY ALARM
OUT       M01562	// L_3rd SPK Y HOME COMPLETE
; L63
LOAD      D001100.8	// L_3rd SPK Y ¢¯©ªA¢®¢¯I¡¤a
OUTP      M01563	// L_3rd SPK Y HOME PLS
; L64
LOAD      M01563	// L_3rd SPK Y HOME PLS
OR        M01564	// L_3rd SPK Y INITIAL HOLD
AND       D001100.8	// L_3rd SPK Y ¢¯©ªA¢®¢¯I¡¤a
AND NOT   M03060	// -
AND NOT   M01565	// L_3rd SPK Y INITIAL ->
OUT       M01564	// L_3rd SPK Y INITIAL HOLD
TON       T0406 5	// L_3rd SPK Y GOINIT->
; L66
LOAD      T0406	// L_3rd SPK Y GOINIT->
OR        M01565	// L_3rd SPK Y INITIAL ->
AND       T0706	// L_3rd SPK Y READY 2s
AND NOT   M02061	// T)L_3rd SPK Y JOG-
AND NOT   M02062	// T)L_3rd SPK Y JOG+
OUT       M01565	// L_3rd SPK Y INITIAL ->

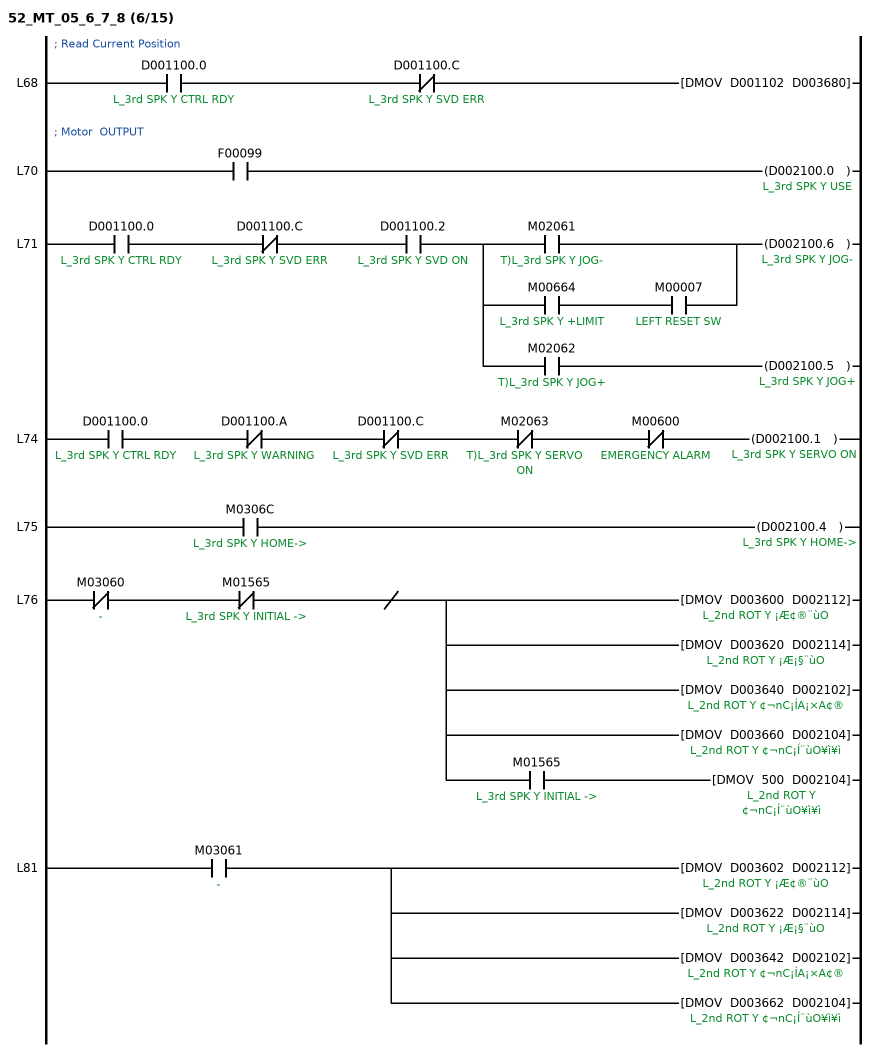
; L68
LOAD      D001100.0	// L_3rd SPK Y CTRL RDY
AND NOT   D001100.C	// L_3rd SPK Y SVD ERR
DMOV      D001102 D003680
// output comment: Read Current Position
//  Motor  OUTPUT
; L70
LOAD      F00099
OUT       D002100.0	// L_3rd SPK Y USE
; L71
LOAD      D001100.0	// L_3rd SPK Y CTRL RDY
AND NOT   D001100.C	// L_3rd SPK Y SVD ERR
AND       D001100.2	// L_3rd SPK Y SVD ON
MPUSH
LOAD      M02061	// T)L_3rd SPK Y JOG-
LOAD      M00664	// L_3rd SPK Y +LIMIT
AND       M00007	// LEFT RESET SW
OR LOAD
AND LOAD
OUT       D002100.6	// L_3rd SPK Y JOG-
MPOP
AND       M02062	// T)L_3rd SPK Y JOG+
OUT       D002100.5	// L_3rd SPK Y JOG+
; L74
LOAD      D001100.0	// L_3rd SPK Y CTRL RDY
AND NOT   D001100.A	// L_3rd SPK Y WARNING
AND NOT   D001100.C	// L_3rd SPK Y SVD ERR
AND NOT   M02063	// T)L_3rd SPK Y SERVO ON
AND NOT   M00600	// EMERGENCY ALARM
OUT       D002100.1	// L_3rd SPK Y SERVO ON
; L75
LOAD      M0306C	// L_3rd SPK Y HOME->
OUT       D002100.4	// L_3rd SPK Y HOME->
; L76
LOAD NOT  M03060	// -
AND NOT   M01565	// L_3rd SPK Y INITIAL ->
NOT
DMOV      D003600 D002112	// L_2nd ROT Y ¡Æ¢®¨ùO
DMOV      D003620 D002114	// L_2nd ROT Y ¡Æ¡§¨ùO
DMOV      D003640 D002102	// L_2nd ROT Y ¢¬nC¡ÍA¡×A¢®
DMOV      D003660 D002104	// L_2nd ROT Y ¢¬nC¡Í¨ùO¥ì¥ì
AND       M01565	// L_3rd SPK Y INITIAL ->
DMOV      500 D002104	// L_2nd ROT Y ¢¬nC¡Í¨ùO¥ì¥ì
; L81
LOAD      M03061	// -
DMOV      D003602 D002112	// L_2nd ROT Y ¡Æ¢®¨ùO
DMOV      D003622 D002114	// L_2nd ROT Y ¡Æ¡§¨ùO
DMOV      D003642 D002102	// L_2nd ROT Y ¢¬nC¡ÍA¡×A¢®
DMOV      D003662 D002104	// L_2nd ROT Y ¢¬nC¡Í¨ùO¥ì¥ì

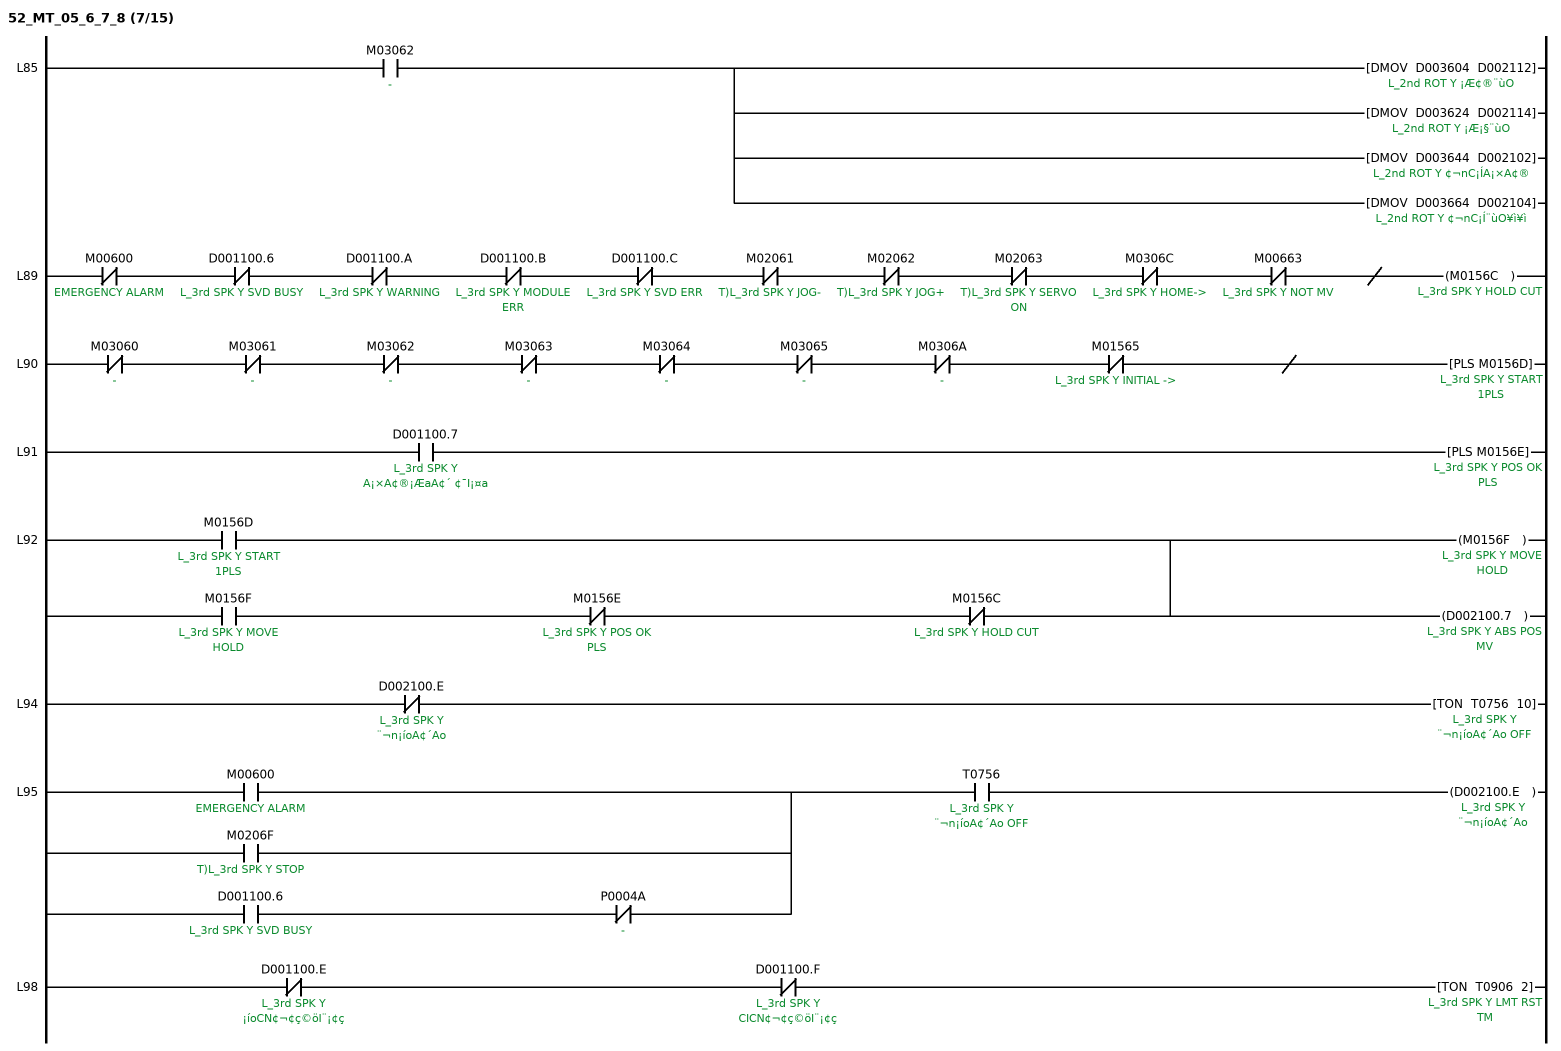
; L85
LOAD      M03062	// -
DMOV      D003604 D002112	// L_2nd ROT Y ¡Æ¢®¨ùO
DMOV      D003624 D002114	// L_2nd ROT Y ¡Æ¡§¨ùO
DMOV      D003644 D002102	// L_2nd ROT Y ¢¬nC¡ÍA¡×A¢®
DMOV      D003664 D002104	// L_2nd ROT Y ¢¬nC¡Í¨ùO¥ì¥ì
; L89
LOAD NOT  M00600	// EMERGENCY ALARM
AND NOT   D001100.6	// L_3rd SPK Y SVD BUSY
AND NOT   D001100.A	// L_3rd SPK Y WARNING
AND NOT   D001100.B	// L_3rd SPK Y MODULE ERR
AND NOT   D001100.C	// L_3rd SPK Y SVD ERR
AND NOT   M02061	// T)L_3rd SPK Y JOG-
AND NOT   M02062	// T)L_3rd SPK Y JOG+
AND NOT   M02063	// T)L_3rd SPK Y SERVO ON
AND NOT   M0306C	// L_3rd SPK Y HOME->
AND NOT   M00663	// L_3rd SPK Y NOT MV
NOT
OUT       M0156C	// L_3rd SPK Y HOLD CUT
; L90
LOAD NOT  M03060	// -
AND NOT   M03061	// -
AND NOT   M03062	// -
AND NOT   M03063	// -
AND NOT   M03064	// -
AND NOT   M03065	// -
AND NOT   M0306A	// -
AND NOT   M01565	// L_3rd SPK Y INITIAL ->
NOT
OUTP      M0156D	// L_3rd SPK Y START 1PLS
; L91
LOAD      D001100.7	// L_3rd SPK Y A¡×A¢®¡ÆaA¢´ ¢¯I¡¤a
OUTP      M0156E	// L_3rd SPK Y POS OK PLS
; L92
LOAD      M0156D	// L_3rd SPK Y START 1PLS
LOAD      M0156F	// L_3rd SPK Y MOVE HOLD
AND NOT   M0156E	// L_3rd SPK Y POS OK PLS
AND NOT   M0156C	// L_3rd SPK Y HOLD CUT
OR LOAD
OUT       M0156F	// L_3rd SPK Y MOVE HOLD
OUT       D002100.7	// L_3rd SPK Y ABS POS MV
; L94
LOAD NOT  D002100.E	// L_3rd SPK Y ¨¬n¡íoA¢´Ao
TON       T0756 10	// L_3rd SPK Y ¨¬n¡íoA¢´Ao OFF
; L95
LOAD      M00600	// EMERGENCY ALARM
OR        M0206F	// T)L_3rd SPK Y STOP
LOAD      D001100.6	// L_3rd SPK Y SVD BUSY
AND NOT   P0004A	// -
OR LOAD
AND       T0756	// L_3rd SPK Y ¨¬n¡íoA¢´Ao OFF
OUT       D002100.E	// L_3rd SPK Y ¨¬n¡íoA¢´Ao
; L98
LOAD NOT  D001100.E	// L_3rd SPK Y ¡íoCN¢¬¢ç©öI¨¡¢ç
AND NOT   D001100.F	// L_3rd SPK Y CICN¢¬¢ç©öI¨¡¢ç
TON       T0906 2	// L_3rd SPK Y LMT RST TM

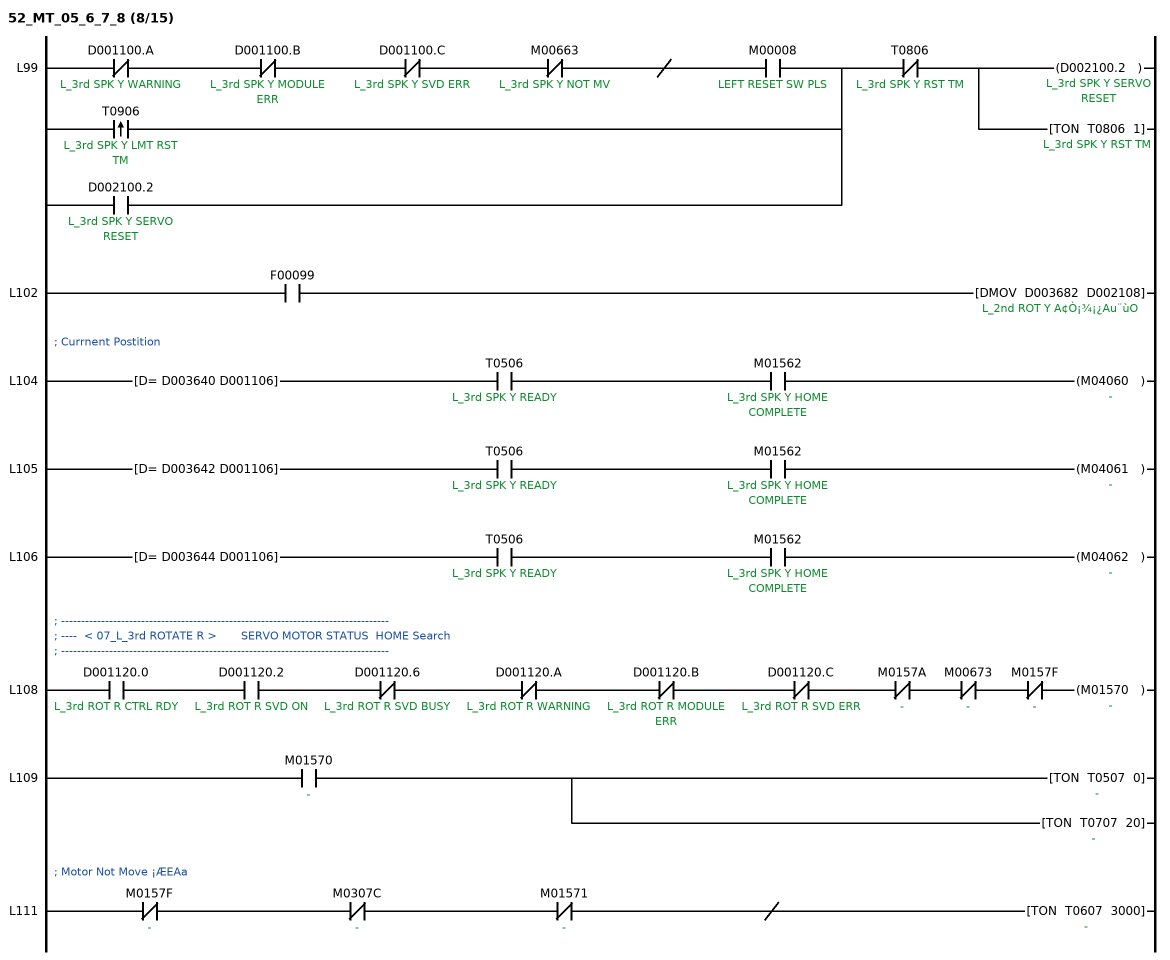
; L99
LOAD NOT  D001100.A	// L_3rd SPK Y WARNING
AND NOT   D001100.B	// L_3rd SPK Y MODULE ERR
AND NOT   D001100.C	// L_3rd SPK Y SVD ERR
AND NOT   M00663	// L_3rd SPK Y NOT MV
NOT
AND       M00008	// LEFT RESET SW PLS
ORP       T0906	// L_3rd SPK Y LMT RST TM
OR        D002100.2	// L_3rd SPK Y SERVO RESET
AND NOT   T0806	// L_3rd SPK Y RST TM
OUT       D002100.2	// L_3rd SPK Y SERVO RESET
TON       T0806 1	// L_3rd SPK Y RST TM
; L102
LOAD      F00099
DMOV      D003682 D002108	// L_2nd ROT Y A¢Ò¡¾¡¿Au¨ùO
// Currnent Postition
; L104
LOADD=    D003640 D001106
AND       T0506	// L_3rd SPK Y READY
AND       M01562	// L_3rd SPK Y HOME COMPLETE
OUT       M04060	// -
; L105
LOADD=    D003642 D001106
AND       T0506	// L_3rd SPK Y READY
AND       M01562	// L_3rd SPK Y HOME COMPLETE
OUT       M04061	// -
; L106
LOADD=    D003644 D001106
AND       T0506	// L_3rd SPK Y READY
AND       M01562	// L_3rd SPK Y HOME COMPLETE
OUT       M04062	// -
// ----------------------------------------------------------------------------------
// 
// ----  < 07_L_3rd ROTATE R >       SERVO MOTOR STATUS  HOME Search
// 
// ----------------------------------------------------------------------------------
; L108
LOAD      D001120.0	// L_3rd ROT R CTRL RDY
AND       D001120.2	// L_3rd ROT R SVD ON
AND NOT   D001120.6	// L_3rd ROT R SVD BUSY
AND NOT   D001120.A	// L_3rd ROT R WARNING
AND NOT   D001120.B	// L_3rd ROT R MODULE ERR
AND NOT   D001120.C	// L_3rd ROT R SVD ERR
AND NOT   M0157A	// -
AND NOT   M00673	// -
AND NOT   M0157F	// -
OUT       M01570	// -
; L109
LOAD      M01570	// -
TON       T0507 0	// -
TON       T0707 20	// -
; L111
LOAD NOT  M0157F	// -
AND NOT   M0307C	// -
AND NOT   M01571	// -
NOT
TON       T0607 3000	// -
// output comment: Motor Not Move ¡ÆEAa

